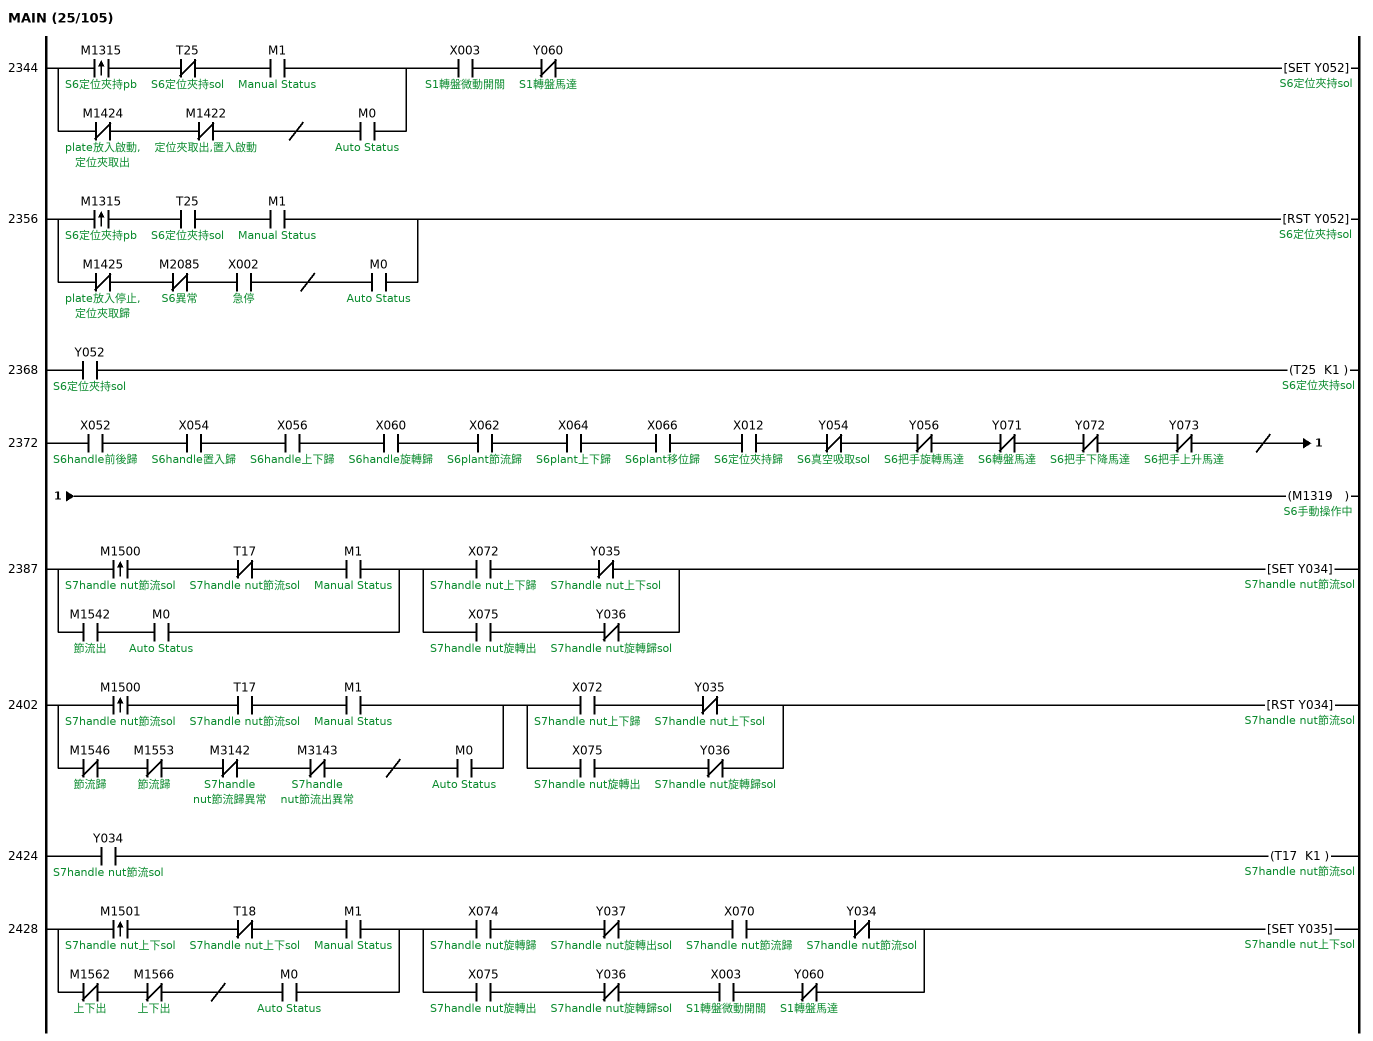
[picture p24: ladder of MAIN, rungs at steps 2344 to 2428]
2344  LDP     M1315  ; S6定位夾持pb
      ANI     T25  ; S6定位夾持sol
      AND     M1  ; Manual Status
      LDI     M1424  ; plate放入啟動,定位夾取出
      ANI     M1422  ; 定位夾取出,置入啟動
      INV
      AND     M0  ; Auto Status
      ORB
      AND     X003  ; S1轉盤微動開關
      ANI     Y060  ; S1轉盤馬達
      SET     Y052  ; S6定位夾持sol
2356  LDP     M1315  ; S6定位夾持pb
      AND     T25  ; S6定位夾持sol
      AND     M1  ; Manual Status
      LDI     M1425  ; plate放入停止,定位夾取歸
      ANI     M2085  ; S6異常
      AND     X002  ; 急停
      INV
      AND     M0  ; Auto Status
      ORB
      RST     Y052  ; S6定位夾持sol
2368  LD      Y052  ; S6定位夾持sol
      OUT     T25 K1  ; S6定位夾持sol
2372  LD      X052  ; S6handle前後歸
      AND     X054  ; S6handle置入歸
      AND     X056  ; S6handle上下歸
      AND     X060  ; S6handle旋轉歸
      AND     X062  ; S6plant節流歸
      AND     X064  ; S6plant上下歸
      AND     X066  ; S6plant移位歸
      AND     X012  ; S6定位夾持歸
      ANI     Y054  ; S6真空吸取sol
      ANI     Y056  ; S6把手旋轉馬達
      ANI     Y071  ; S6轉盤馬達
      ANI     Y072  ; S6把手下降馬達
      ANI     Y073  ; S6把手上升馬達
      INV
      OUT     M1319  ; S6手動操作中
2387  LDP     M1500  ; S7handle nut節流sol
      ANI     T17  ; S7handle nut節流sol
      AND     M1  ; Manual Status
      LD      M1542  ; 節流出
      AND     M0  ; Auto Status
      ORB
      LD      X072  ; S7handle nut上下歸
      ANI     Y035  ; S7handle nut上下sol
      LD      X075  ; S7handle nut旋轉出
      ANI     Y036  ; S7handle nut旋轉歸sol
      ORB
      ANB
      SET     Y034  ; S7handle nut節流sol
2402  LDP     M1500  ; S7handle nut節流sol
      AND     T17  ; S7handle nut節流sol
      AND     M1  ; Manual Status
      LDI     M1546  ; 節流歸
      ANI     M1553  ; 節流歸
      ANI     M3142  ; S7handle nut節流歸異常
      ANI     M3143  ; S7handle nut節流出異常
      INV
      AND     M0  ; Auto Status
      ORB
      LD      X072  ; S7handle nut上下歸
      ANI     Y035  ; S7handle nut上下sol
      LD      X075  ; S7handle nut旋轉出
      ANI     Y036  ; S7handle nut旋轉歸sol
      ORB
      ANB
      RST     Y034  ; S7handle nut節流sol
2424  LD      Y034  ; S7handle nut節流sol
      OUT     T17 K1  ; S7handle nut節流sol
2428  LDP     M1501  ; S7handle nut上下sol
      ANI     T18  ; S7handle nut上下sol
      AND     M1  ; Manual Status
      LDI     M1562  ; 上下出
      ANI     M1566  ; 上下出
      INV
      AND     M0  ; Auto Status
      ORB
      LD      X074  ; S7handle nut旋轉歸
      ANI     Y037  ; S7handle nut旋轉出sol
      AND     X070  ; S7handle nut節流歸
      ANI     Y034  ; S7handle nut節流sol
      LD      X075  ; S7handle nut旋轉出
      ANI     Y036  ; S7handle nut旋轉歸sol
      AND     X003  ; S1轉盤微動開關
      ANI     Y060  ; S1轉盤馬達
      ORB
      ANB
      SET     Y035  ; S7handle nut上下sol
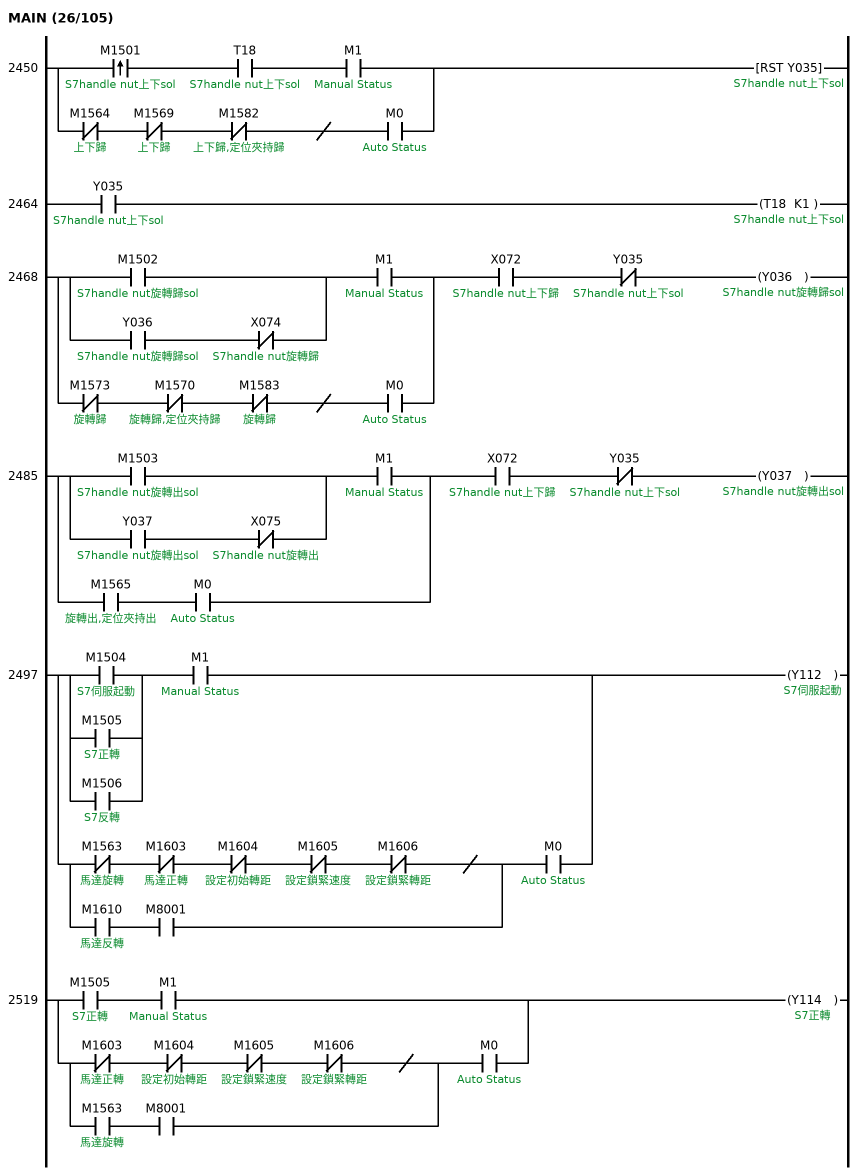
2450  LDP     M1501  ; S7handle nut上下sol
      AND     T18  ; S7handle nut上下sol
      AND     M1  ; Manual Status
      LDI     M1564  ; 上下歸
      ANI     M1569  ; 上下歸
      ANI     M1582  ; 上下歸,定位夾持歸
      INV
      AND     M0  ; Auto Status
      ORB
      RST     Y035  ; S7handle nut上下sol
2464  LD      Y035  ; S7handle nut上下sol
      OUT     T18 K1  ; S7handle nut上下sol
2468  LD      M1502  ; S7handle nut旋轉歸sol
      LD      Y036  ; S7handle nut旋轉歸sol
      ANI     X074  ; S7handle nut旋轉歸
      ORB
      AND     M1  ; Manual Status
      LDI     M1573  ; 旋轉歸
      ANI     M1570  ; 旋轉歸,定位夾持歸
      ANI     M1583  ; 旋轉歸
      INV
      AND     M0  ; Auto Status
      ORB
      AND     X072  ; S7handle nut上下歸
      ANI     Y035  ; S7handle nut上下sol
      OUT     Y036  ; S7handle nut旋轉歸sol
2485  LD      M1503  ; S7handle nut旋轉出sol
      LD      Y037  ; S7handle nut旋轉出sol
      ANI     X075  ; S7handle nut旋轉出
      ORB
      AND     M1  ; Manual Status
      LD      M1565  ; 旋轉出,定位夾持出
      AND     M0  ; Auto Status
      ORB
      AND     X072  ; S7handle nut上下歸
      ANI     Y035  ; S7handle nut上下sol
      OUT     Y037  ; S7handle nut旋轉出sol
2497  LD      M1504  ; S7伺服起動
      OR      M1505  ; S7正轉
      OR      M1506  ; S7反轉
      AND     M1  ; Manual Status
      LDI     M1563  ; 馬達旋轉
      ANI     M1603  ; 馬達正轉
      ANI     M1604  ; 設定初始轉距
      ANI     M1605  ; 設定鎖緊速度
      ANI     M1606  ; 設定鎖緊轉距
      INV
      LD      M1610  ; 馬達反轉
      AND     M8001
      ORB
      AND     M0  ; Auto Status
      ORB
      OUT     Y112  ; S7伺服起動
2519  LD      M1505  ; S7正轉
      AND     M1  ; Manual Status
      LDI     M1603  ; 馬達正轉
      ANI     M1604  ; 設定初始轉距
      ANI     M1605  ; 設定鎖緊速度
      ANI     M1606  ; 設定鎖緊轉距
      INV
      LD      M1563  ; 馬達旋轉
      AND     M8001
      ORB
      AND     M0  ; Auto Status
      ORB
      OUT     Y114  ; S7正轉
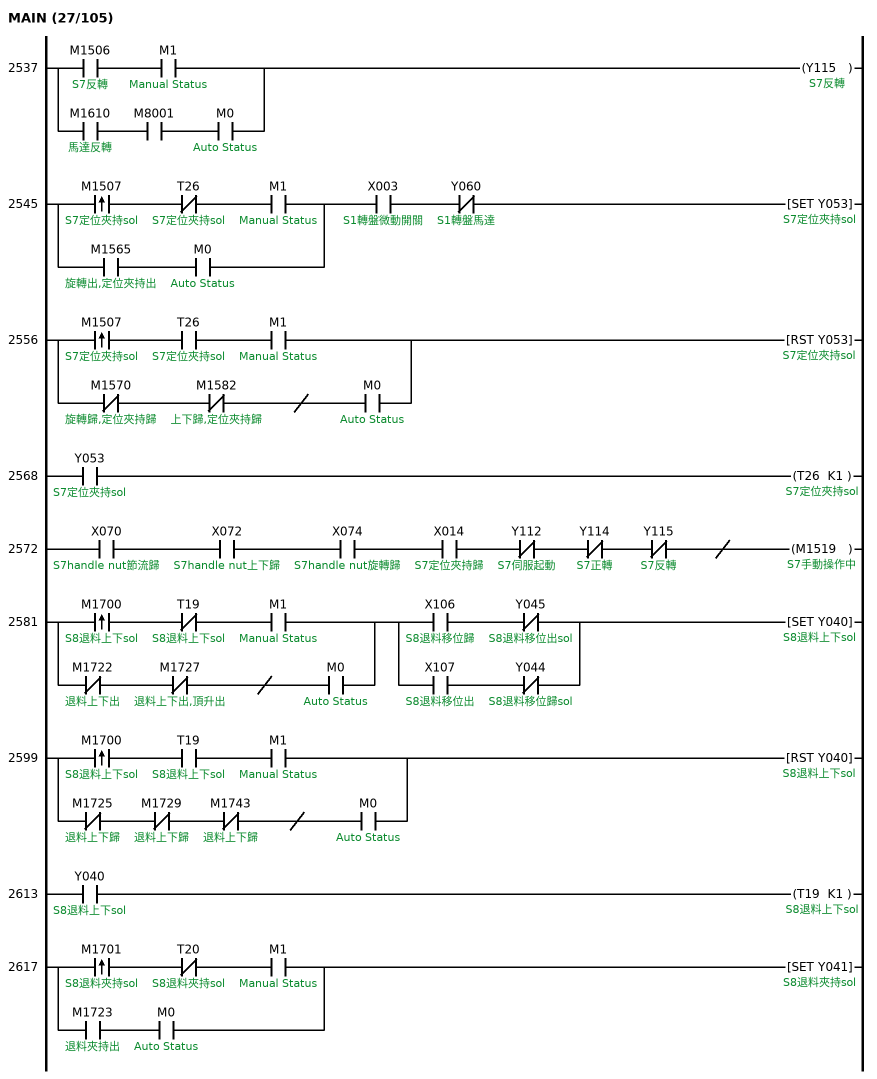
2537  LD      M1506  ; S7反轉
      AND     M1  ; Manual Status
      LD      M1610  ; 馬達反轉
      AND     M8001
      AND     M0  ; Auto Status
      ORB
      OUT     Y115  ; S7反轉
2545  LDP     M1507  ; S7定位夾持sol
      ANI     T26  ; S7定位夾持sol
      AND     M1  ; Manual Status
      LD      M1565  ; 旋轉出,定位夾持出
      AND     M0  ; Auto Status
      ORB
      AND     X003  ; S1轉盤微動開關
      ANI     Y060  ; S1轉盤馬達
      SET     Y053  ; S7定位夾持sol
2556  LDP     M1507  ; S7定位夾持sol
      AND     T26  ; S7定位夾持sol
      AND     M1  ; Manual Status
      LDI     M1570  ; 旋轉歸,定位夾持歸
      ANI     M1582  ; 上下歸,定位夾持歸
      INV
      AND     M0  ; Auto Status
      ORB
      RST     Y053  ; S7定位夾持sol
2568  LD      Y053  ; S7定位夾持sol
      OUT     T26 K1  ; S7定位夾持sol
2572  LD      X070  ; S7handle nut節流歸
      AND     X072  ; S7handle nut上下歸
      AND     X074  ; S7handle nut旋轉歸
      AND     X014  ; S7定位夾持歸
      ANI     Y112  ; S7伺服起動
      ANI     Y114  ; S7正轉
      ANI     Y115  ; S7反轉
      INV
      OUT     M1519  ; S7手動操作中
2581  LDP     M1700  ; S8退料上下sol
      ANI     T19  ; S8退料上下sol
      AND     M1  ; Manual Status
      LDI     M1722  ; 退料上下出
      ANI     M1727  ; 退料上下出,頂升出
      INV
      AND     M0  ; Auto Status
      ORB
      LD      X106  ; S8退料移位歸
      ANI     Y045  ; S8退料移位出sol
      LD      X107  ; S8退料移位出
      ANI     Y044  ; S8退料移位歸sol
      ORB
      ANB
      SET     Y040  ; S8退料上下sol
2599  LDP     M1700  ; S8退料上下sol
      AND     T19  ; S8退料上下sol
      AND     M1  ; Manual Status
      LDI     M1725  ; 退料上下歸
      ANI     M1729  ; 退料上下歸
      ANI     M1743  ; 退料上下歸
      INV
      AND     M0  ; Auto Status
      ORB
      RST     Y040  ; S8退料上下sol
2613  LD      Y040  ; S8退料上下sol
      OUT     T19 K1  ; S8退料上下sol
2617  LDP     M1701  ; S8退料夾持sol
      ANI     T20  ; S8退料夾持sol
      AND     M1  ; Manual Status
      LD      M1723  ; 退料夾持出
      AND     M0  ; Auto Status
      ORB
      SET     Y041  ; S8退料夾持sol
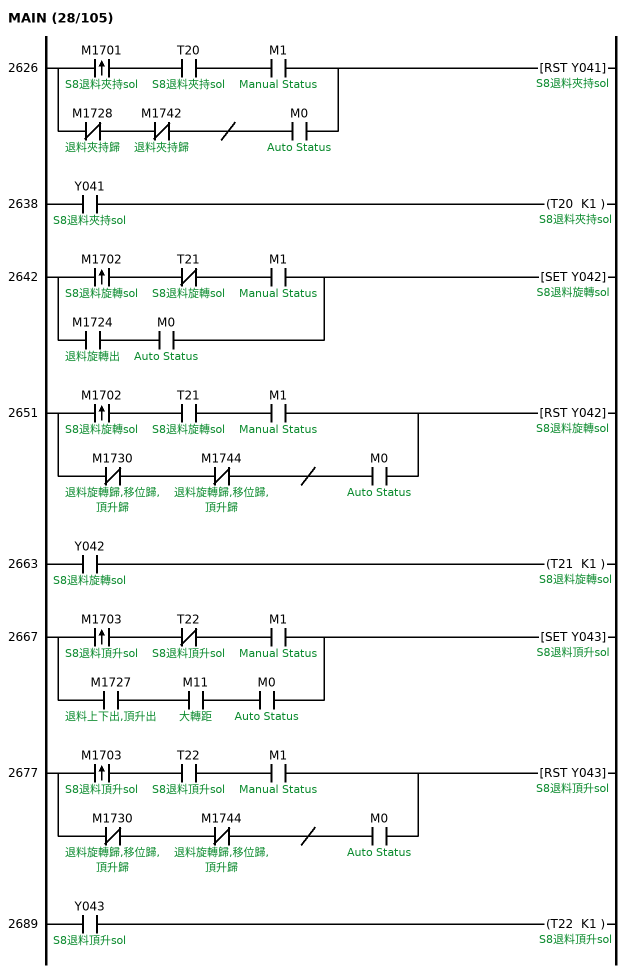
2626  LDP     M1701  ; S8退料夾持sol
      AND     T20  ; S8退料夾持sol
      AND     M1  ; Manual Status
      LDI     M1728  ; 退料夾持歸
      ANI     M1742  ; 退料夾持歸
      INV
      AND     M0  ; Auto Status
      ORB
      RST     Y041  ; S8退料夾持sol
2638  LD      Y041  ; S8退料夾持sol
      OUT     T20 K1  ; S8退料夾持sol
2642  LDP     M1702  ; S8退料旋轉sol
      ANI     T21  ; S8退料旋轉sol
      AND     M1  ; Manual Status
      LD      M1724  ; 退料旋轉出
      AND     M0  ; Auto Status
      ORB
      SET     Y042  ; S8退料旋轉sol
2651  LDP     M1702  ; S8退料旋轉sol
      AND     T21  ; S8退料旋轉sol
      AND     M1  ; Manual Status
      LDI     M1730  ; 退料旋轉歸,移位歸,頂升歸
      ANI     M1744  ; 退料旋轉歸,移位歸,頂升歸
      INV
      AND     M0  ; Auto Status
      ORB
      RST     Y042  ; S8退料旋轉sol
2663  LD      Y042  ; S8退料旋轉sol
      OUT     T21 K1  ; S8退料旋轉sol
2667  LDP     M1703  ; S8退料頂升sol
      ANI     T22  ; S8退料頂升sol
      AND     M1  ; Manual Status
      LD      M1727  ; 退料上下出,頂升出
      AND     M11  ; 大轉距
      AND     M0  ; Auto Status
      ORB
      SET     Y043  ; S8退料頂升sol
2677  LDP     M1703  ; S8退料頂升sol
      AND     T22  ; S8退料頂升sol
      AND     M1  ; Manual Status
      LDI     M1730  ; 退料旋轉歸,移位歸,頂升歸
      ANI     M1744  ; 退料旋轉歸,移位歸,頂升歸
      INV
      AND     M0  ; Auto Status
      ORB
      RST     Y043  ; S8退料頂升sol
2689  LD      Y043  ; S8退料頂升sol
      OUT     T22 K1  ; S8退料頂升sol
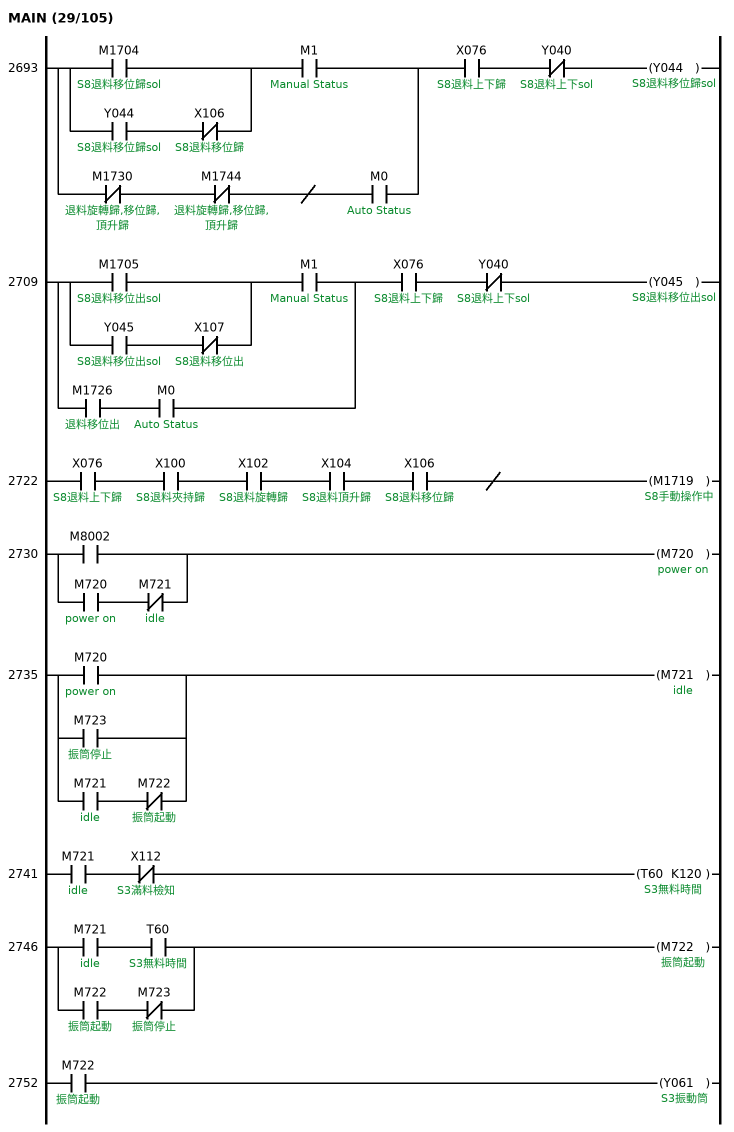
2693  LD      M1704  ; S8退料移位歸sol
      LD      Y044  ; S8退料移位歸sol
      ANI     X106  ; S8退料移位歸
      ORB
      AND     M1  ; Manual Status
      LDI     M1730  ; 退料旋轉歸,移位歸,頂升歸
      ANI     M1744  ; 退料旋轉歸,移位歸,頂升歸
      INV
      AND     M0  ; Auto Status
      ORB
      AND     X076  ; S8退料上下歸
      ANI     Y040  ; S8退料上下sol
      OUT     Y044  ; S8退料移位歸sol
2709  LD      M1705  ; S8退料移位出sol
      LD      Y045  ; S8退料移位出sol
      ANI     X107  ; S8退料移位出
      ORB
      AND     M1  ; Manual Status
      LD      M1726  ; 退料移位出
      AND     M0  ; Auto Status
      ORB
      AND     X076  ; S8退料上下歸
      ANI     Y040  ; S8退料上下sol
      OUT     Y045  ; S8退料移位出sol
2722  LD      X076  ; S8退料上下歸
      AND     X100  ; S8退料夾持歸
      AND     X102  ; S8退料旋轉歸
      AND     X104  ; S8退料頂升歸
      AND     X106  ; S8退料移位歸
      INV
      OUT     M1719  ; S8手動操作中
2730  LD      M8002
      LD      M720  ; power on
      ANI     M721  ; idle
      ORB
      OUT     M720  ; power on
2735  LD      M720  ; power on
      OR      M723  ; 振筒停止
      LD      M721  ; idle
      ANI     M722  ; 振筒起動
      ORB
      OUT     M721  ; idle
2741  LD      M721  ; idle
      ANI     X112  ; S3滿料檢知
      OUT     T60 K120  ; S3無料時間
2746  LD      M721  ; idle
      AND     T60  ; S3無料時間
      LD      M722  ; 振筒起動
      ANI     M723  ; 振筒停止
      ORB
      OUT     M722  ; 振筒起動
2752  LD      M722  ; 振筒起動
      OUT     Y061  ; S3振動筒
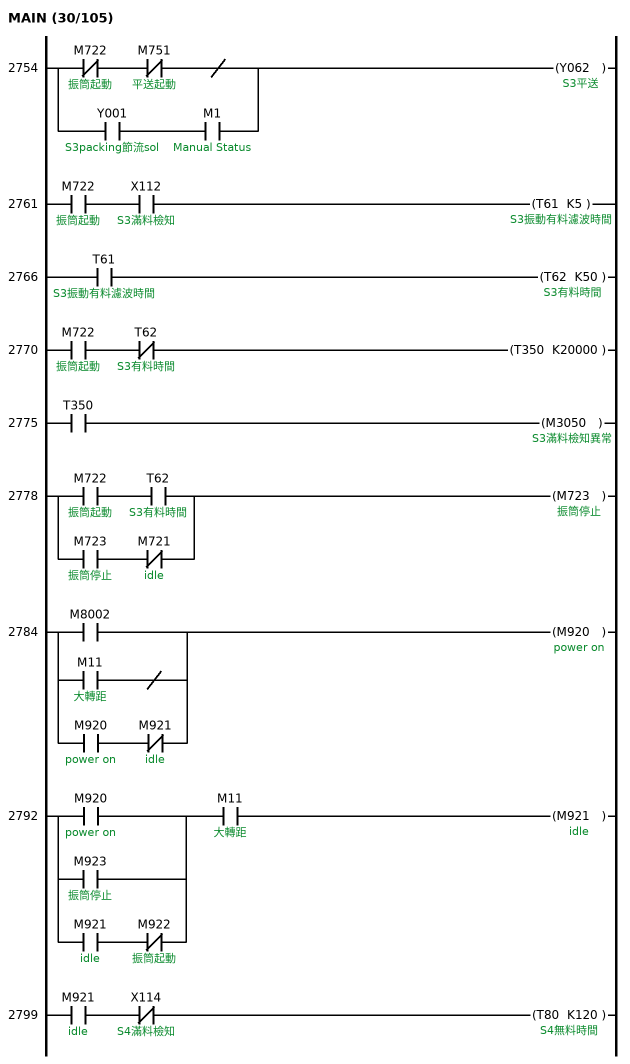
2754  LDI     M722  ; 振筒起動
      ANI     M751  ; 平送起動
      INV
      LD      Y001  ; S3packing節流sol
      AND     M1  ; Manual Status
      ORB
      OUT     Y062  ; S3平送
2761  LD      M722  ; 振筒起動
      AND     X112  ; S3滿料檢知
      OUT     T61 K5  ; S3振動有料濾波時間
2766  LD      T61  ; S3振動有料濾波時間
      OUT     T62 K50  ; S3有料時間
2770  LD      M722  ; 振筒起動
      ANI     T62  ; S3有料時間
      OUT     T350 K20000
2775  LD      T350
      OUT     M3050  ; S3滿料檢知異常
2778  LD      M722  ; 振筒起動
      AND     T62  ; S3有料時間
      LD      M723  ; 振筒停止
      ANI     M721  ; idle
      ORB
      OUT     M723  ; 振筒停止
2784  LD      M8002
      LD      M11  ; 大轉距
      INV
      ORB
      LD      M920  ; power on
      ANI     M921  ; idle
      ORB
      OUT     M920  ; power on
2792  LD      M920  ; power on
      OR      M923  ; 振筒停止
      LD      M921  ; idle
      ANI     M922  ; 振筒起動
      ORB
      AND     M11  ; 大轉距
      OUT     M921  ; idle
2799  LD      M921  ; idle
      ANI     X114  ; S4滿料檢知
      OUT     T80 K120  ; S4無料時間
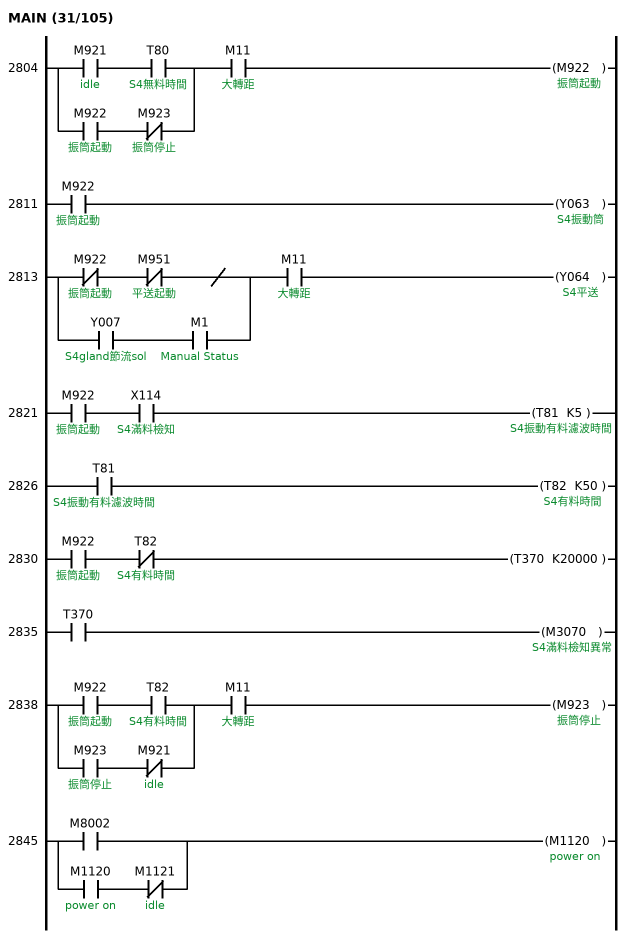
2804  LD      M921  ; idle
      AND     T80  ; S4無料時間
      LD      M922  ; 振筒起動
      ANI     M923  ; 振筒停止
      ORB
      AND     M11  ; 大轉距
      OUT     M922  ; 振筒起動
2811  LD      M922  ; 振筒起動
      OUT     Y063  ; S4振動筒
2813  LDI     M922  ; 振筒起動
      ANI     M951  ; 平送起動
      INV
      LD      Y007  ; S4gland節流sol
      AND     M1  ; Manual Status
      ORB
      AND     M11  ; 大轉距
      OUT     Y064  ; S4平送
2821  LD      M922  ; 振筒起動
      AND     X114  ; S4滿料檢知
      OUT     T81 K5  ; S4振動有料濾波時間
2826  LD      T81  ; S4振動有料濾波時間
      OUT     T82 K50  ; S4有料時間
2830  LD      M922  ; 振筒起動
      ANI     T82  ; S4有料時間
      OUT     T370 K20000
2835  LD      T370
      OUT     M3070  ; S4滿料檢知異常
2838  LD      M922  ; 振筒起動
      AND     T82  ; S4有料時間
      LD      M923  ; 振筒停止
      ANI     M921  ; idle
      ORB
      AND     M11  ; 大轉距
      OUT     M923  ; 振筒停止
2845  LD      M8002
      LD      M1120  ; power on
      ANI     M1121  ; idle
      ORB
      OUT     M1120  ; power on
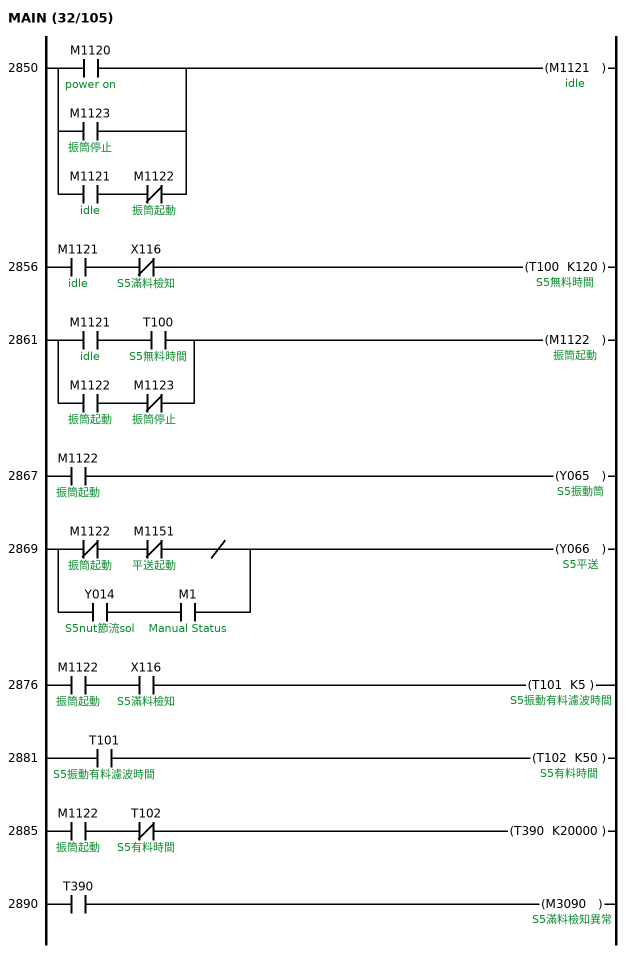
2850  LD      M1120  ; power on
      OR      M1123  ; 振筒停止
      LD      M1121  ; idle
      ANI     M1122  ; 振筒起動
      ORB
      OUT     M1121  ; idle
2856  LD      M1121  ; idle
      ANI     X116  ; S5滿料檢知
      OUT     T100 K120  ; S5無料時間
2861  LD      M1121  ; idle
      AND     T100  ; S5無料時間
      LD      M1122  ; 振筒起動
      ANI     M1123  ; 振筒停止
      ORB
      OUT     M1122  ; 振筒起動
2867  LD      M1122  ; 振筒起動
      OUT     Y065  ; S5振動筒
2869  LDI     M1122  ; 振筒起動
      ANI     M1151  ; 平送起動
      INV
      LD      Y014  ; S5nut節流sol
      AND     M1  ; Manual Status
      ORB
      OUT     Y066  ; S5平送
2876  LD      M1122  ; 振筒起動
      AND     X116  ; S5滿料檢知
      OUT     T101 K5  ; S5振動有料濾波時間
2881  LD      T101  ; S5振動有料濾波時間
      OUT     T102 K50  ; S5有料時間
2885  LD      M1122  ; 振筒起動
      ANI     T102  ; S5有料時間
      OUT     T390 K20000
2890  LD      T390
      OUT     M3090  ; S5滿料檢知異常
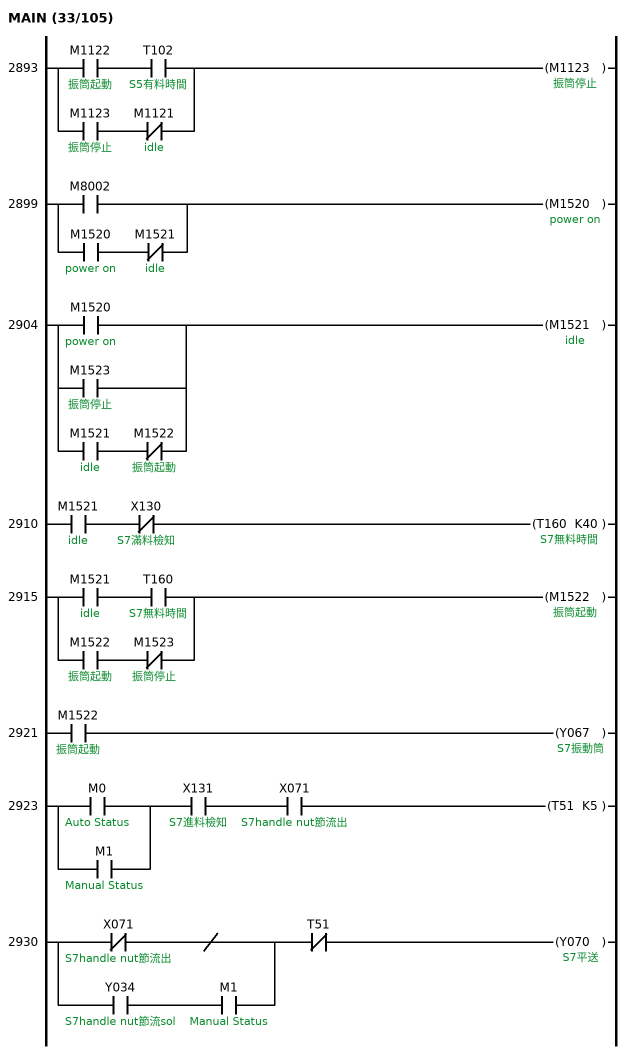
2893  LD      M1122  ; 振筒起動
      AND     T102  ; S5有料時間
      LD      M1123  ; 振筒停止
      ANI     M1121  ; idle
      ORB
      OUT     M1123  ; 振筒停止
2899  LD      M8002
      LD      M1520  ; power on
      ANI     M1521  ; idle
      ORB
      OUT     M1520  ; power on
2904  LD      M1520  ; power on
      OR      M1523  ; 振筒停止
      LD      M1521  ; idle
      ANI     M1522  ; 振筒起動
      ORB
      OUT     M1521  ; idle
2910  LD      M1521  ; idle
      ANI     X130  ; S7滿料檢知
      OUT     T160 K40  ; S7無料時間
2915  LD      M1521  ; idle
      AND     T160  ; S7無料時間
      LD      M1522  ; 振筒起動
      ANI     M1523  ; 振筒停止
      ORB
      OUT     M1522  ; 振筒起動
2921  LD      M1522  ; 振筒起動
      OUT     Y067  ; S7振動筒
2923  LD      M0  ; Auto Status
      OR      M1  ; Manual Status
      AND     X131  ; S7進料檢知
      AND     X071  ; S7handle nut節流出
      OUT     T51 K5
2930  LDI     X071  ; S7handle nut節流出
      INV
      LD      Y034  ; S7handle nut節流sol
      AND     M1  ; Manual Status
      ORB
      ANI     T51
      OUT     Y070  ; S7平送
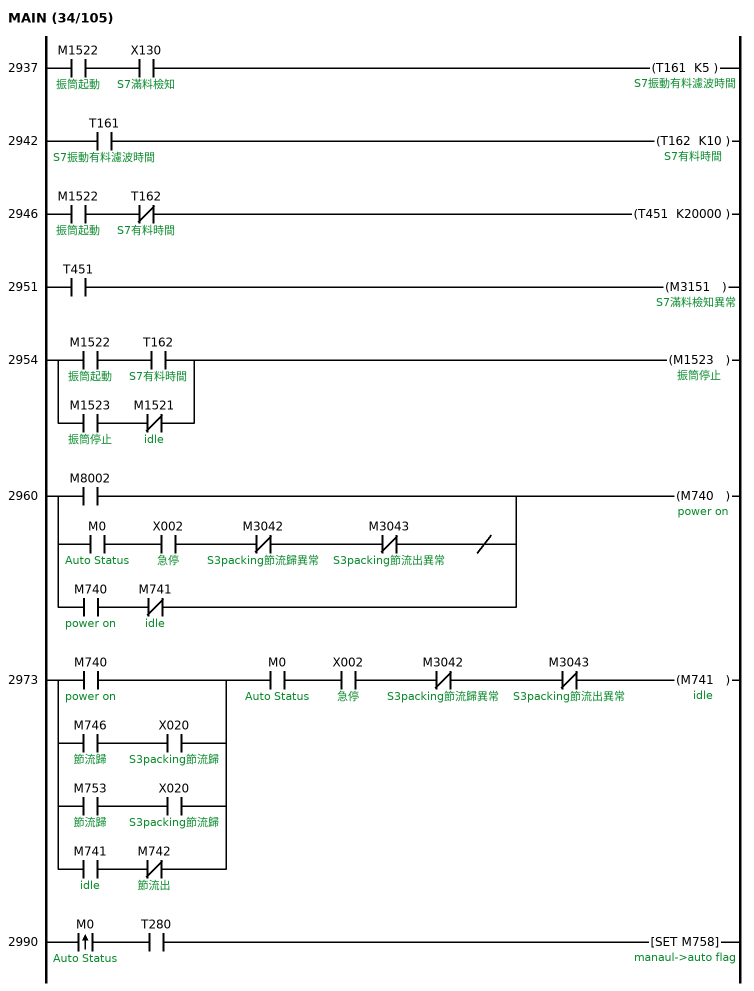
2937  LD      M1522  ; 振筒起動
      AND     X130  ; S7滿料檢知
      OUT     T161 K5  ; S7振動有料濾波時間
2942  LD      T161  ; S7振動有料濾波時間
      OUT     T162 K10  ; S7有料時間
2946  LD      M1522  ; 振筒起動
      ANI     T162  ; S7有料時間
      OUT     T451 K20000
2951  LD      T451
      OUT     M3151  ; S7滿料檢知異常
2954  LD      M1522  ; 振筒起動
      AND     T162  ; S7有料時間
      LD      M1523  ; 振筒停止
      ANI     M1521  ; idle
      ORB
      OUT     M1523  ; 振筒停止
2960  LD      M8002
      LD      M0  ; Auto Status
      AND     X002  ; 急停
      ANI     M3042  ; S3packing節流歸異常
      ANI     M3043  ; S3packing節流出異常
      INV
      ORB
      LD      M740  ; power on
      ANI     M741  ; idle
      ORB
      OUT     M740  ; power on
2973  LD      M740  ; power on
      LD      M746  ; 節流歸
      AND     X020  ; S3packing節流歸
      ORB
      LD      M753  ; 節流歸
      AND     X020  ; S3packing節流歸
      ORB
      LD      M741  ; idle
      ANI     M742  ; 節流出
      ORB
      AND     M0  ; Auto Status
      AND     X002  ; 急停
      ANI     M3042  ; S3packing節流歸異常
      ANI     M3043  ; S3packing節流出異常
      OUT     M741  ; idle
2990  LDP     M0  ; Auto Status
      AND     T280
      SET     M758  ; manaul->auto flag
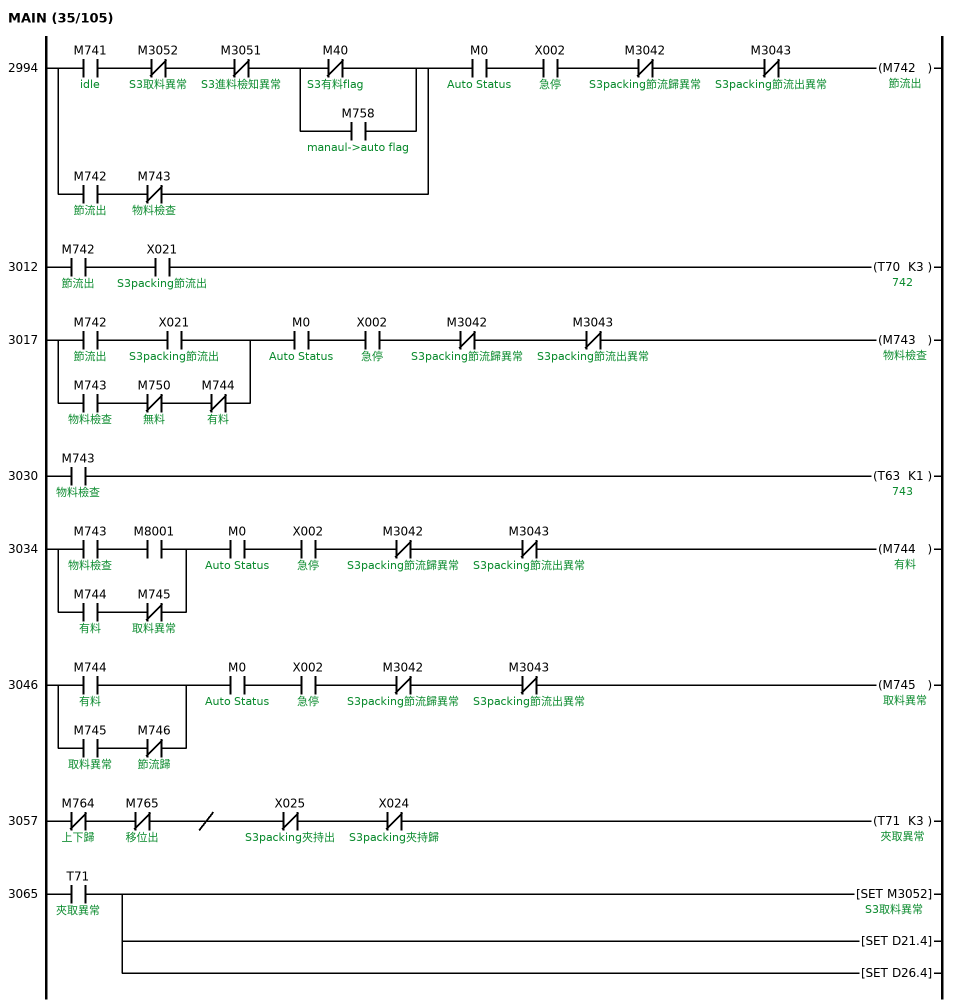
2994  LD      M741  ; idle
      ANI     M3052  ; S3取料異常
      ANI     M3051  ; S3進料檢知異常
      LDI     M40  ; S3有料flag
      OR      M758  ; manaul->auto flag
      ANB
      LD      M742  ; 節流出
      ANI     M743  ; 物料檢查
      ORB
      AND     M0  ; Auto Status
      AND     X002  ; 急停
      ANI     M3042  ; S3packing節流歸異常
      ANI     M3043  ; S3packing節流出異常
      OUT     M742  ; 節流出
3012  LD      M742  ; 節流出
      AND     X021  ; S3packing節流出
      OUT     T70 K3  ; 742
3017  LD      M742  ; 節流出
      AND     X021  ; S3packing節流出
      LD      M743  ; 物料檢查
      ANI     M750  ; 無料
      ANI     M744  ; 有料
      ORB
      AND     M0  ; Auto Status
      AND     X002  ; 急停
      ANI     M3042  ; S3packing節流歸異常
      ANI     M3043  ; S3packing節流出異常
      OUT     M743  ; 物料檢查
3030  LD      M743  ; 物料檢查
      OUT     T63 K1  ; 743
3034  LD      M743  ; 物料檢查
      AND     M8001
      LD      M744  ; 有料
      ANI     M745  ; 取料異常
      ORB
      AND     M0  ; Auto Status
      AND     X002  ; 急停
      ANI     M3042  ; S3packing節流歸異常
      ANI     M3043  ; S3packing節流出異常
      OUT     M744  ; 有料
3046  LD      M744  ; 有料
      LD      M745  ; 取料異常
      ANI     M746  ; 節流歸
      ORB
      AND     M0  ; Auto Status
      AND     X002  ; 急停
      ANI     M3042  ; S3packing節流歸異常
      ANI     M3043  ; S3packing節流出異常
      OUT     M745  ; 取料異常
3057  LDI     M764  ; 上下歸
      ANI     M765  ; 移位出
      INV
      ANI     X025  ; S3packing夾持出
      ANI     X024  ; S3packing夾持歸
      OUT     T71 K3  ; 夾取異常
3065  LD      T71  ; 夾取異常
      SET     M3052  ; S3取料異常
      SET     D21.4
      SET     D26.4
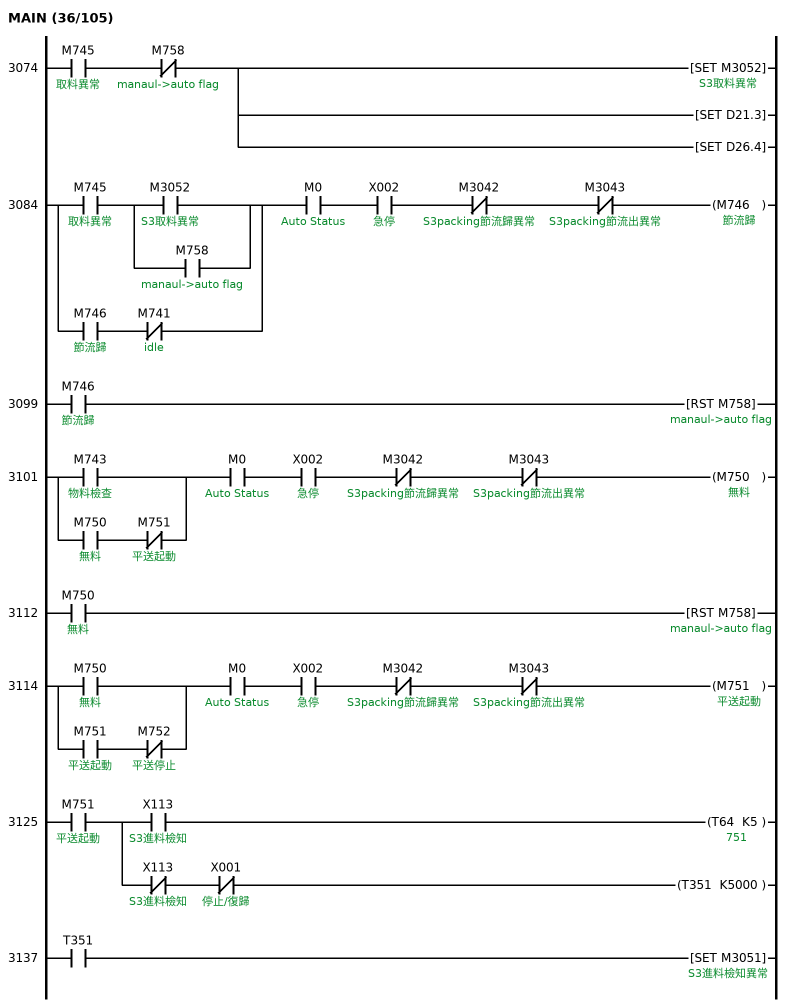
3074  LD      M745  ; 取料異常
      ANI     M758  ; manaul->auto flag
      SET     M3052  ; S3取料異常
      SET     D21.3
      SET     D26.4
3084  LD      M745  ; 取料異常
      LD      M3052  ; S3取料異常
      OR      M758  ; manaul->auto flag
      ANB
      LD      M746  ; 節流歸
      ANI     M741  ; idle
      ORB
      AND     M0  ; Auto Status
      AND     X002  ; 急停
      ANI     M3042  ; S3packing節流歸異常
      ANI     M3043  ; S3packing節流出異常
      OUT     M746  ; 節流歸
3099  LD      M746  ; 節流歸
      RST     M758  ; manaul->auto flag
3101  LD      M743  ; 物料檢查
      LD      M750  ; 無料
      ANI     M751  ; 平送起動
      ORB
      AND     M0  ; Auto Status
      AND     X002  ; 急停
      ANI     M3042  ; S3packing節流歸異常
      ANI     M3043  ; S3packing節流出異常
      OUT     M750  ; 無料
3112  LD      M750  ; 無料
      RST     M758  ; manaul->auto flag
3114  LD      M750  ; 無料
      LD      M751  ; 平送起動
      ANI     M752  ; 平送停止
      ORB
      AND     M0  ; Auto Status
      AND     X002  ; 急停
      ANI     M3042  ; S3packing節流歸異常
      ANI     M3043  ; S3packing節流出異常
      OUT     M751  ; 平送起動
3125  LD      M751  ; 平送起動
      MPS
      AND     X113  ; S3進料檢知
      OUT     T64 K5  ; 751
      MPP
      ANI     X113  ; S3進料檢知
      ANI     X001  ; 停止/復歸
      OUT     T351 K5000
3137  LD      T351
      SET     M3051  ; S3進料檢知異常
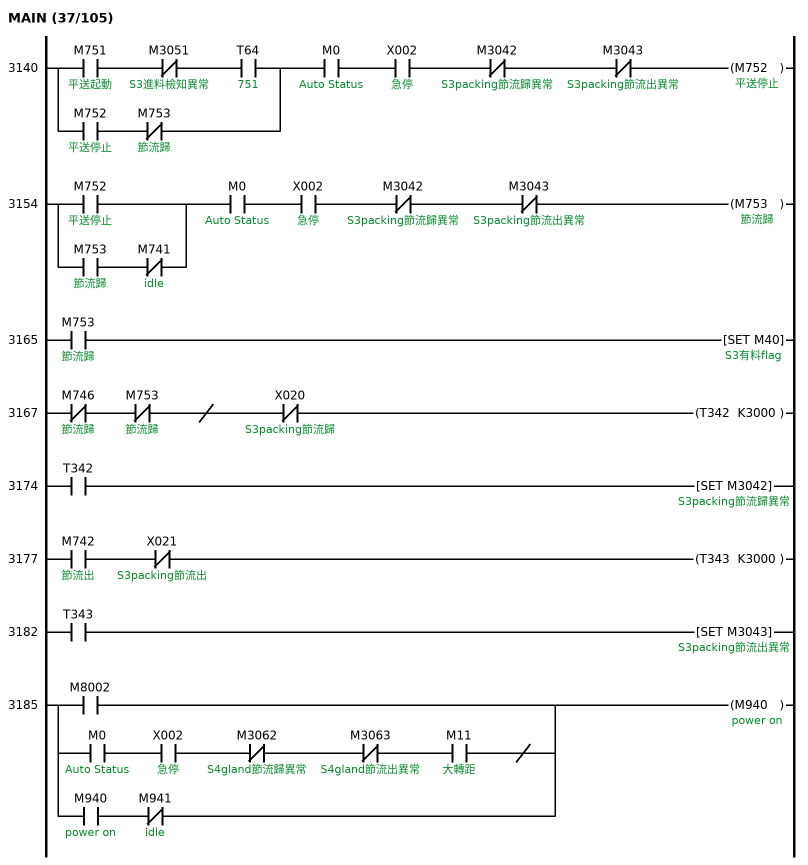
3140  LD      M751  ; 平送起動
      ANI     M3051  ; S3進料檢知異常
      AND     T64  ; 751
      LD      M752  ; 平送停止
      ANI     M753  ; 節流歸
      ORB
      AND     M0  ; Auto Status
      AND     X002  ; 急停
      ANI     M3042  ; S3packing節流歸異常
      ANI     M3043  ; S3packing節流出異常
      OUT     M752  ; 平送停止
3154  LD      M752  ; 平送停止
      LD      M753  ; 節流歸
      ANI     M741  ; idle
      ORB
      AND     M0  ; Auto Status
      AND     X002  ; 急停
      ANI     M3042  ; S3packing節流歸異常
      ANI     M3043  ; S3packing節流出異常
      OUT     M753  ; 節流歸
3165  LD      M753  ; 節流歸
      SET     M40  ; S3有料flag
3167  LDI     M746  ; 節流歸
      ANI     M753  ; 節流歸
      INV
      ANI     X020  ; S3packing節流歸
      OUT     T342 K3000
3174  LD      T342
      SET     M3042  ; S3packing節流歸異常
3177  LD      M742  ; 節流出
      ANI     X021  ; S3packing節流出
      OUT     T343 K3000
3182  LD      T343
      SET     M3043  ; S3packing節流出異常
3185  LD      M8002
      LD      M0  ; Auto Status
      AND     X002  ; 急停
      ANI     M3062  ; S4gland節流歸異常
      ANI     M3063  ; S4gland節流出異常
      AND     M11  ; 大轉距
      INV
      ORB
      LD      M940  ; power on
      ANI     M941  ; idle
      ORB
      OUT     M940  ; power on
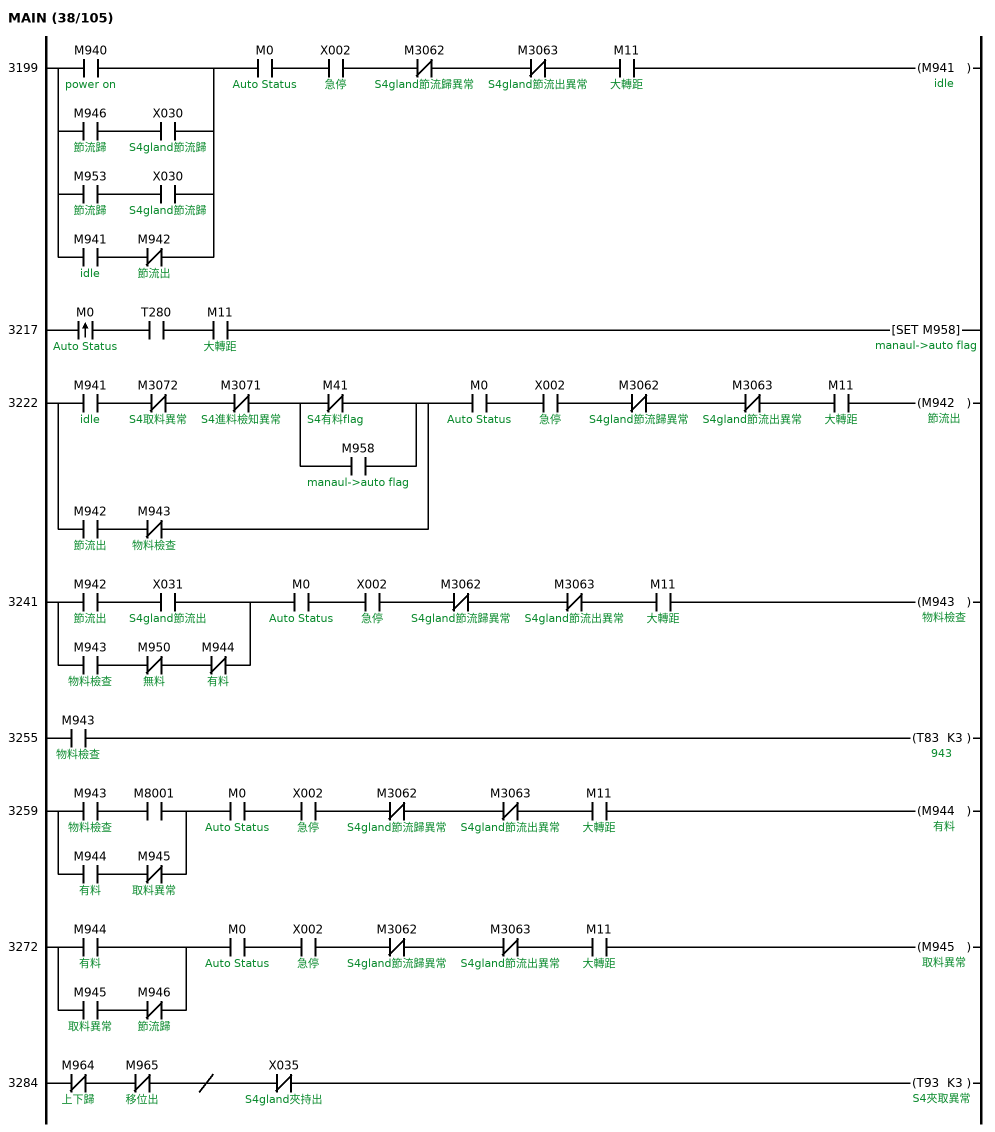
3199  LD      M940  ; power on
      LD      M946  ; 節流歸
      AND     X030  ; S4gland節流歸
      ORB
      LD      M953  ; 節流歸
      AND     X030  ; S4gland節流歸
      ORB
      LD      M941  ; idle
      ANI     M942  ; 節流出
      ORB
      AND     M0  ; Auto Status
      AND     X002  ; 急停
      ANI     M3062  ; S4gland節流歸異常
      ANI     M3063  ; S4gland節流出異常
      AND     M11  ; 大轉距
      OUT     M941  ; idle
3217  LDP     M0  ; Auto Status
      AND     T280
      AND     M11  ; 大轉距
      SET     M958  ; manaul->auto flag
3222  LD      M941  ; idle
      ANI     M3072  ; S4取料異常
      ANI     M3071  ; S4進料檢知異常
      LDI     M41  ; S4有料flag
      OR      M958  ; manaul->auto flag
      ANB
      LD      M942  ; 節流出
      ANI     M943  ; 物料檢查
      ORB
      AND     M0  ; Auto Status
      AND     X002  ; 急停
      ANI     M3062  ; S4gland節流歸異常
      ANI     M3063  ; S4gland節流出異常
      AND     M11  ; 大轉距
      OUT     M942  ; 節流出
3241  LD      M942  ; 節流出
      AND     X031  ; S4gland節流出
      LD      M943  ; 物料檢查
      ANI     M950  ; 無料
      ANI     M944  ; 有料
      ORB
      AND     M0  ; Auto Status
      AND     X002  ; 急停
      ANI     M3062  ; S4gland節流歸異常
      ANI     M3063  ; S4gland節流出異常
      AND     M11  ; 大轉距
      OUT     M943  ; 物料檢查
3255  LD      M943  ; 物料檢查
      OUT     T83 K3  ; 943
3259  LD      M943  ; 物料檢查
      AND     M8001
      LD      M944  ; 有料
      ANI     M945  ; 取料異常
      ORB
      AND     M0  ; Auto Status
      AND     X002  ; 急停
      ANI     M3062  ; S4gland節流歸異常
      ANI     M3063  ; S4gland節流出異常
      AND     M11  ; 大轉距
      OUT     M944  ; 有料
3272  LD      M944  ; 有料
      LD      M945  ; 取料異常
      ANI     M946  ; 節流歸
      ORB
      AND     M0  ; Auto Status
      AND     X002  ; 急停
      ANI     M3062  ; S4gland節流歸異常
      ANI     M3063  ; S4gland節流出異常
      AND     M11  ; 大轉距
      OUT     M945  ; 取料異常
3284  LDI     M964  ; 上下歸
      ANI     M965  ; 移位出
      INV
      ANI     X035  ; S4gland夾持出
      OUT     T93 K3  ; S4夾取異常
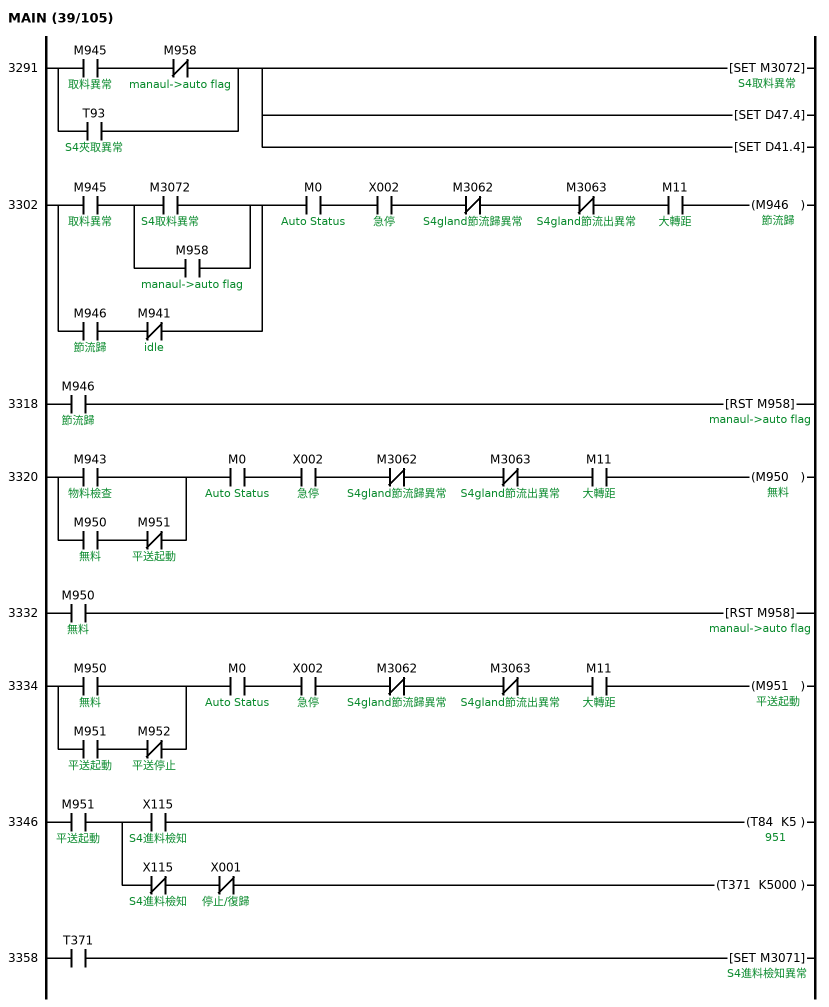
3291  LD      M945  ; 取料異常
      ANI     M958  ; manaul->auto flag
      OR      T93  ; S4夾取異常
      SET     M3072  ; S4取料異常
      SET     D47.4
      SET     D41.4
3302  LD      M945  ; 取料異常
      LD      M3072  ; S4取料異常
      OR      M958  ; manaul->auto flag
      ANB
      LD      M946  ; 節流歸
      ANI     M941  ; idle
      ORB
      AND     M0  ; Auto Status
      AND     X002  ; 急停
      ANI     M3062  ; S4gland節流歸異常
      ANI     M3063  ; S4gland節流出異常
      AND     M11  ; 大轉距
      OUT     M946  ; 節流歸
3318  LD      M946  ; 節流歸
      RST     M958  ; manaul->auto flag
3320  LD      M943  ; 物料檢查
      LD      M950  ; 無料
      ANI     M951  ; 平送起動
      ORB
      AND     M0  ; Auto Status
      AND     X002  ; 急停
      ANI     M3062  ; S4gland節流歸異常
      ANI     M3063  ; S4gland節流出異常
      AND     M11  ; 大轉距
      OUT     M950  ; 無料
3332  LD      M950  ; 無料
      RST     M958  ; manaul->auto flag
3334  LD      M950  ; 無料
      LD      M951  ; 平送起動
      ANI     M952  ; 平送停止
      ORB
      AND     M0  ; Auto Status
      AND     X002  ; 急停
      ANI     M3062  ; S4gland節流歸異常
      ANI     M3063  ; S4gland節流出異常
      AND     M11  ; 大轉距
      OUT     M951  ; 平送起動
3346  LD      M951  ; 平送起動
      MPS
      AND     X115  ; S4進料檢知
      OUT     T84 K5  ; 951
      MPP
      ANI     X115  ; S4進料檢知
      ANI     X001  ; 停止/復歸
      OUT     T371 K5000
3358  LD      T371
      SET     M3071  ; S4進料檢知異常
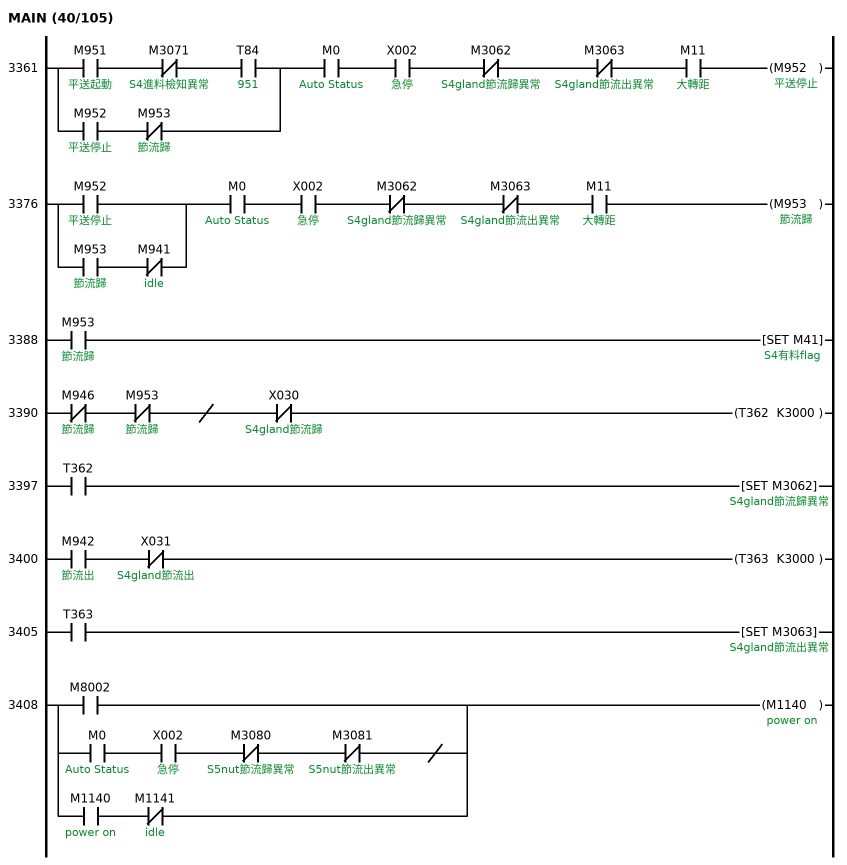
3361  LD      M951  ; 平送起動
      ANI     M3071  ; S4進料檢知異常
      AND     T84  ; 951
      LD      M952  ; 平送停止
      ANI     M953  ; 節流歸
      ORB
      AND     M0  ; Auto Status
      AND     X002  ; 急停
      ANI     M3062  ; S4gland節流歸異常
      ANI     M3063  ; S4gland節流出異常
      AND     M11  ; 大轉距
      OUT     M952  ; 平送停止
3376  LD      M952  ; 平送停止
      LD      M953  ; 節流歸
      ANI     M941  ; idle
      ORB
      AND     M0  ; Auto Status
      AND     X002  ; 急停
      ANI     M3062  ; S4gland節流歸異常
      ANI     M3063  ; S4gland節流出異常
      AND     M11  ; 大轉距
      OUT     M953  ; 節流歸
3388  LD      M953  ; 節流歸
      SET     M41  ; S4有料flag
3390  LDI     M946  ; 節流歸
      ANI     M953  ; 節流歸
      INV
      ANI     X030  ; S4gland節流歸
      OUT     T362 K3000
3397  LD      T362
      SET     M3062  ; S4gland節流歸異常
3400  LD      M942  ; 節流出
      ANI     X031  ; S4gland節流出
      OUT     T363 K3000
3405  LD      T363
      SET     M3063  ; S4gland節流出異常
3408  LD      M8002
      LD      M0  ; Auto Status
      AND     X002  ; 急停
      ANI     M3080  ; S5nut節流歸異常
      ANI     M3081  ; S5nut節流出異常
      INV
      ORB
      LD      M1140  ; power on
      ANI     M1141  ; idle
      ORB
      OUT     M1140  ; power on
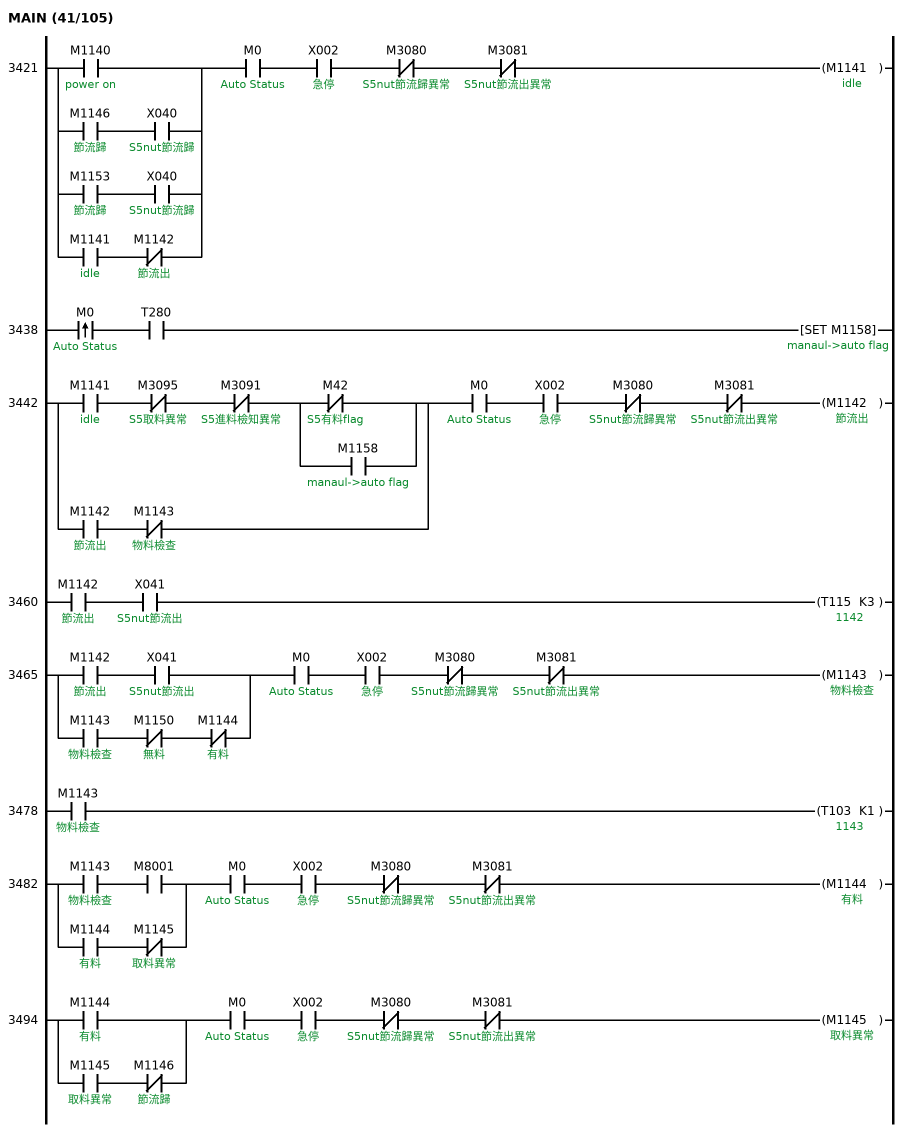
3421  LD      M1140  ; power on
      LD      M1146  ; 節流歸
      AND     X040  ; S5nut節流歸
      ORB
      LD      M1153  ; 節流歸
      AND     X040  ; S5nut節流歸
      ORB
      LD      M1141  ; idle
      ANI     M1142  ; 節流出
      ORB
      AND     M0  ; Auto Status
      AND     X002  ; 急停
      ANI     M3080  ; S5nut節流歸異常
      ANI     M3081  ; S5nut節流出異常
      OUT     M1141  ; idle
3438  LDP     M0  ; Auto Status
      AND     T280
      SET     M1158  ; manaul->auto flag
3442  LD      M1141  ; idle
      ANI     M3095  ; S5取料異常
      ANI     M3091  ; S5進料檢知異常
      LDI     M42  ; S5有料flag
      OR      M1158  ; manaul->auto flag
      ANB
      LD      M1142  ; 節流出
      ANI     M1143  ; 物料檢查
      ORB
      AND     M0  ; Auto Status
      AND     X002  ; 急停
      ANI     M3080  ; S5nut節流歸異常
      ANI     M3081  ; S5nut節流出異常
      OUT     M1142  ; 節流出
3460  LD      M1142  ; 節流出
      AND     X041  ; S5nut節流出
      OUT     T115 K3  ; 1142
3465  LD      M1142  ; 節流出
      AND     X041  ; S5nut節流出
      LD      M1143  ; 物料檢查
      ANI     M1150  ; 無料
      ANI     M1144  ; 有料
      ORB
      AND     M0  ; Auto Status
      AND     X002  ; 急停
      ANI     M3080  ; S5nut節流歸異常
      ANI     M3081  ; S5nut節流出異常
      OUT     M1143  ; 物料檢查
3478  LD      M1143  ; 物料檢查
      OUT     T103 K1  ; 1143
3482  LD      M1143  ; 物料檢查
      AND     M8001
      LD      M1144  ; 有料
      ANI     M1145  ; 取料異常
      ORB
      AND     M0  ; Auto Status
      AND     X002  ; 急停
      ANI     M3080  ; S5nut節流歸異常
      ANI     M3081  ; S5nut節流出異常
      OUT     M1144  ; 有料
3494  LD      M1144  ; 有料
      LD      M1145  ; 取料異常
      ANI     M1146  ; 節流歸
      ORB
      AND     M0  ; Auto Status
      AND     X002  ; 急停
      ANI     M3080  ; S5nut節流歸異常
      ANI     M3081  ; S5nut節流出異常
      OUT     M1145  ; 取料異常
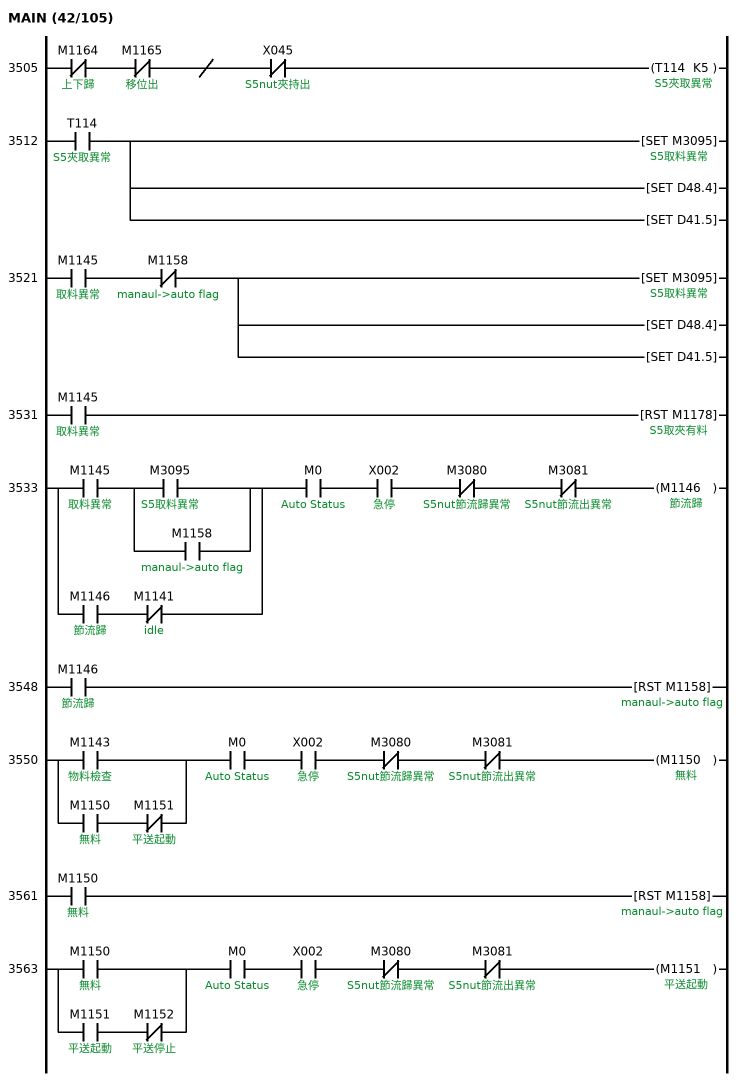
3505  LDI     M1164  ; 上下歸
      ANI     M1165  ; 移位出
      INV
      ANI     X045  ; S5nut夾持出
      OUT     T114 K5  ; S5夾取異常
3512  LD      T114  ; S5夾取異常
      SET     M3095  ; S5取料異常
      SET     D48.4
      SET     D41.5
3521  LD      M1145  ; 取料異常
      ANI     M1158  ; manaul->auto flag
      SET     M3095  ; S5取料異常
      SET     D48.4
      SET     D41.5
3531  LD      M1145  ; 取料異常
      RST     M1178  ; S5取夾有料
3533  LD      M1145  ; 取料異常
      LD      M3095  ; S5取料異常
      OR      M1158  ; manaul->auto flag
      ANB
      LD      M1146  ; 節流歸
      ANI     M1141  ; idle
      ORB
      AND     M0  ; Auto Status
      AND     X002  ; 急停
      ANI     M3080  ; S5nut節流歸異常
      ANI     M3081  ; S5nut節流出異常
      OUT     M1146  ; 節流歸
3548  LD      M1146  ; 節流歸
      RST     M1158  ; manaul->auto flag
3550  LD      M1143  ; 物料檢查
      LD      M1150  ; 無料
      ANI     M1151  ; 平送起動
      ORB
      AND     M0  ; Auto Status
      AND     X002  ; 急停
      ANI     M3080  ; S5nut節流歸異常
      ANI     M3081  ; S5nut節流出異常
      OUT     M1150  ; 無料
3561  LD      M1150  ; 無料
      RST     M1158  ; manaul->auto flag
3563  LD      M1150  ; 無料
      LD      M1151  ; 平送起動
      ANI     M1152  ; 平送停止
      ORB
      AND     M0  ; Auto Status
      AND     X002  ; 急停
      ANI     M3080  ; S5nut節流歸異常
      ANI     M3081  ; S5nut節流出異常
      OUT     M1151  ; 平送起動
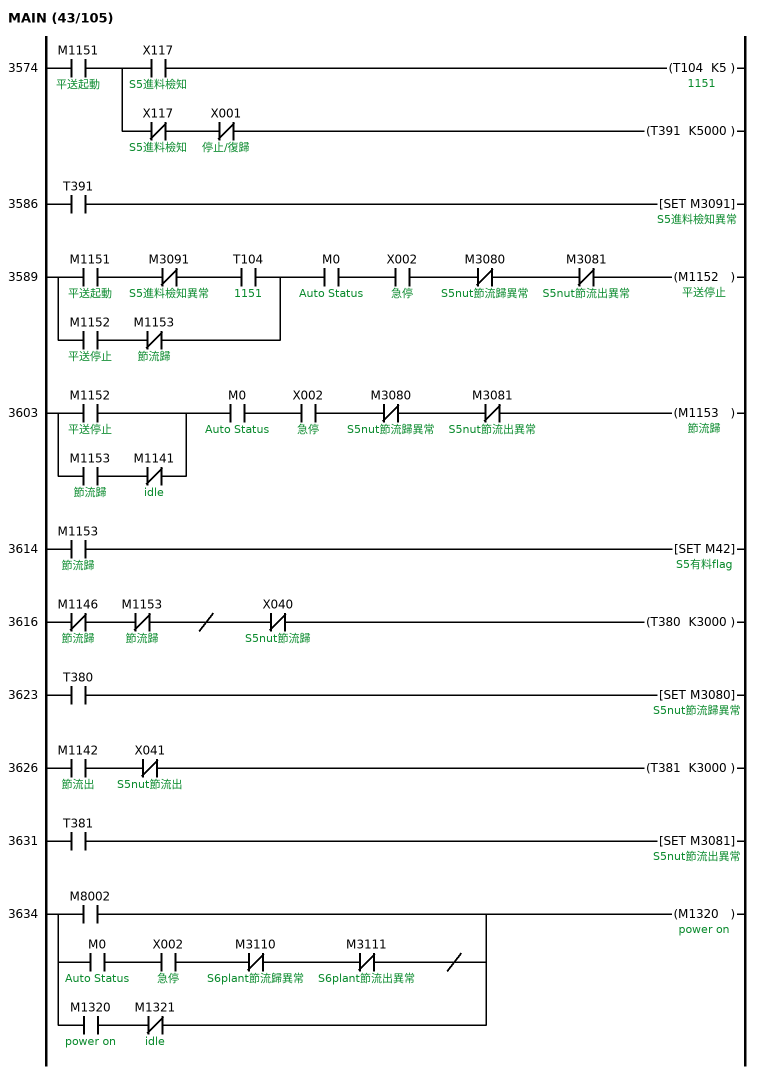
3574  LD      M1151  ; 平送起動
      MPS
      AND     X117  ; S5進料檢知
      OUT     T104 K5  ; 1151
      MPP
      ANI     X117  ; S5進料檢知
      ANI     X001  ; 停止/復歸
      OUT     T391 K5000
3586  LD      T391
      SET     M3091  ; S5進料檢知異常
3589  LD      M1151  ; 平送起動
      ANI     M3091  ; S5進料檢知異常
      AND     T104  ; 1151
      LD      M1152  ; 平送停止
      ANI     M1153  ; 節流歸
      ORB
      AND     M0  ; Auto Status
      AND     X002  ; 急停
      ANI     M3080  ; S5nut節流歸異常
      ANI     M3081  ; S5nut節流出異常
      OUT     M1152  ; 平送停止
3603  LD      M1152  ; 平送停止
      LD      M1153  ; 節流歸
      ANI     M1141  ; idle
      ORB
      AND     M0  ; Auto Status
      AND     X002  ; 急停
      ANI     M3080  ; S5nut節流歸異常
      ANI     M3081  ; S5nut節流出異常
      OUT     M1153  ; 節流歸
3614  LD      M1153  ; 節流歸
      SET     M42  ; S5有料flag
3616  LDI     M1146  ; 節流歸
      ANI     M1153  ; 節流歸
      INV
      ANI     X040  ; S5nut節流歸
      OUT     T380 K3000
3623  LD      T380
      SET     M3080  ; S5nut節流歸異常
3626  LD      M1142  ; 節流出
      ANI     X041  ; S5nut節流出
      OUT     T381 K3000
3631  LD      T381
      SET     M3081  ; S5nut節流出異常
3634  LD      M8002
      LD      M0  ; Auto Status
      AND     X002  ; 急停
      ANI     M3110  ; S6plant節流歸異常
      ANI     M3111  ; S6plant節流出異常
      INV
      ORB
      LD      M1320  ; power on
      ANI     M1321  ; idle
      ORB
      OUT     M1320  ; power on
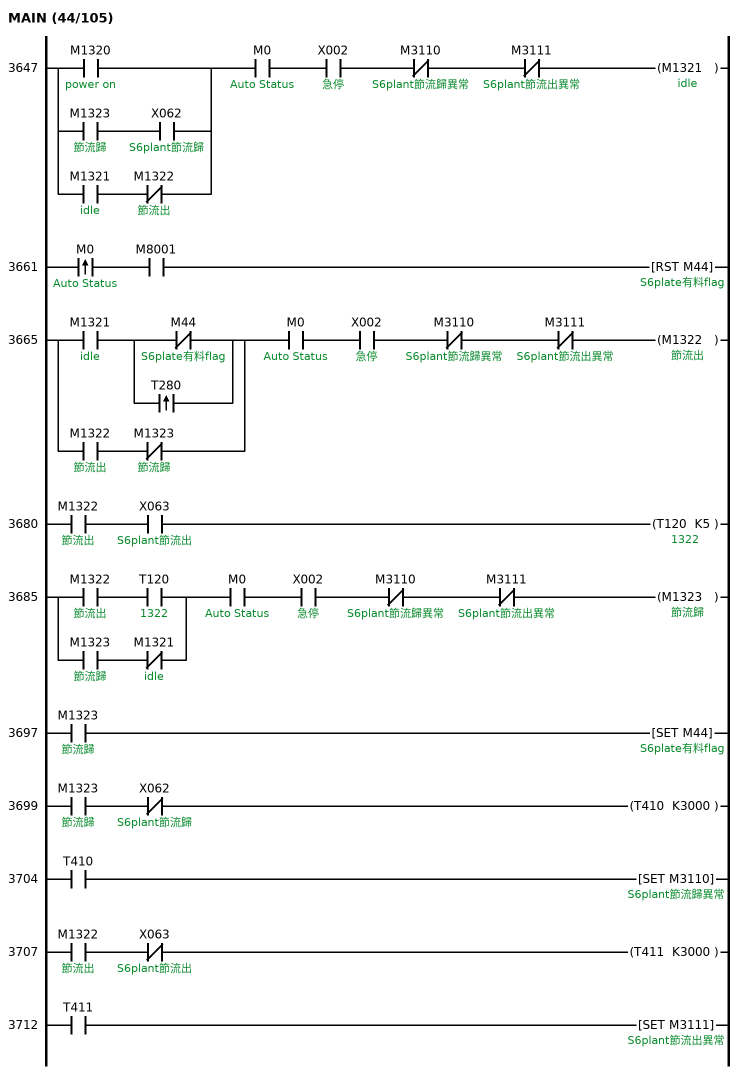
3647  LD      M1320  ; power on
      LD      M1323  ; 節流歸
      AND     X062  ; S6plant節流歸
      ORB
      LD      M1321  ; idle
      ANI     M1322  ; 節流出
      ORB
      AND     M0  ; Auto Status
      AND     X002  ; 急停
      ANI     M3110  ; S6plant節流歸異常
      ANI     M3111  ; S6plant節流出異常
      OUT     M1321  ; idle
3661  LDP     M0  ; Auto Status
      AND     M8001
      RST     M44  ; S6plate有料flag
3665  LD      M1321  ; idle
      LDI     M44  ; S6plate有料flag
      ORP     T280
      ANB
      LD      M1322  ; 節流出
      ANI     M1323  ; 節流歸
      ORB
      AND     M0  ; Auto Status
      AND     X002  ; 急停
      ANI     M3110  ; S6plant節流歸異常
      ANI     M3111  ; S6plant節流出異常
      OUT     M1322  ; 節流出
3680  LD      M1322  ; 節流出
      AND     X063  ; S6plant節流出
      OUT     T120 K5  ; 1322
3685  LD      M1322  ; 節流出
      AND     T120  ; 1322
      LD      M1323  ; 節流歸
      ANI     M1321  ; idle
      ORB
      AND     M0  ; Auto Status
      AND     X002  ; 急停
      ANI     M3110  ; S6plant節流歸異常
      ANI     M3111  ; S6plant節流出異常
      OUT     M1323  ; 節流歸
3697  LD      M1323  ; 節流歸
      SET     M44  ; S6plate有料flag
3699  LD      M1323  ; 節流歸
      ANI     X062  ; S6plant節流歸
      OUT     T410 K3000
3704  LD      T410
      SET     M3110  ; S6plant節流歸異常
3707  LD      M1322  ; 節流出
      ANI     X063  ; S6plant節流出
      OUT     T411 K3000
3712  LD      T411
      SET     M3111  ; S6plant節流出異常
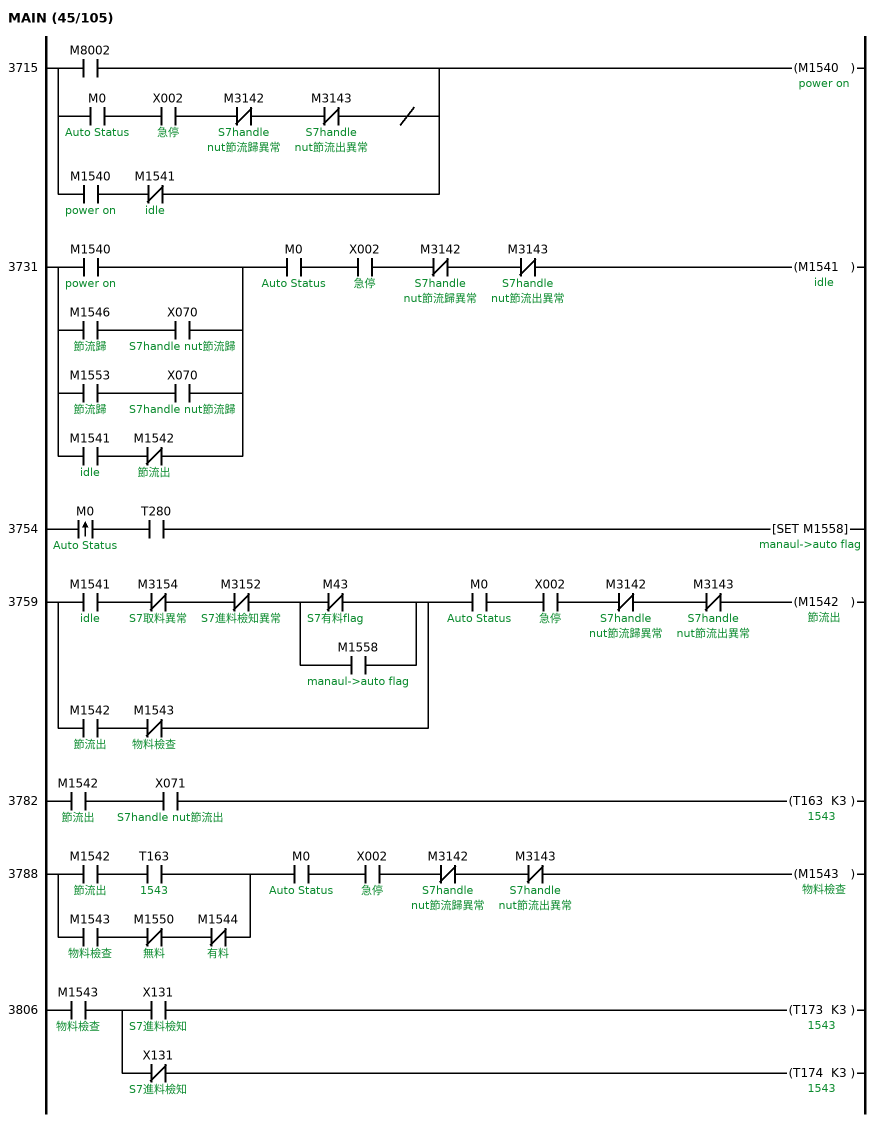
3715  LD      M8002
      LD      M0  ; Auto Status
      AND     X002  ; 急停
      ANI     M3142  ; S7handle nut節流歸異常
      ANI     M3143  ; S7handle nut節流出異常
      INV
      ORB
      LD      M1540  ; power on
      ANI     M1541  ; idle
      ORB
      OUT     M1540  ; power on
3731  LD      M1540  ; power on
      LD      M1546  ; 節流歸
      AND     X070  ; S7handle nut節流歸
      ORB
      LD      M1553  ; 節流歸
      AND     X070  ; S7handle nut節流歸
      ORB
      LD      M1541  ; idle
      ANI     M1542  ; 節流出
      ORB
      AND     M0  ; Auto Status
      AND     X002  ; 急停
      ANI     M3142  ; S7handle nut節流歸異常
      ANI     M3143  ; S7handle nut節流出異常
      OUT     M1541  ; idle
3754  LDP     M0  ; Auto Status
      AND     T280
      SET     M1558  ; manaul->auto flag
3759  LD      M1541  ; idle
      ANI     M3154  ; S7取料異常
      ANI     M3152  ; S7進料檢知異常
      LDI     M43  ; S7有料flag
      OR      M1558  ; manaul->auto flag
      ANB
      LD      M1542  ; 節流出
      ANI     M1543  ; 物料檢查
      ORB
      AND     M0  ; Auto Status
      AND     X002  ; 急停
      ANI     M3142  ; S7handle nut節流歸異常
      ANI     M3143  ; S7handle nut節流出異常
      OUT     M1542  ; 節流出
3782  LD      M1542  ; 節流出
      AND     X071  ; S7handle nut節流出
      OUT     T163 K3  ; 1543
3788  LD      M1542  ; 節流出
      AND     T163  ; 1543
      LD      M1543  ; 物料檢查
      ANI     M1550  ; 無料
      ANI     M1544  ; 有料
      ORB
      AND     M0  ; Auto Status
      AND     X002  ; 急停
      ANI     M3142  ; S7handle nut節流歸異常
      ANI     M3143  ; S7handle nut節流出異常
      OUT     M1543  ; 物料檢查
3806  LD      M1543  ; 物料檢查
      MPS
      AND     X131  ; S7進料檢知
      OUT     T173 K3  ; 1543
      MPP
      ANI     X131  ; S7進料檢知
      OUT     T174 K3  ; 1543
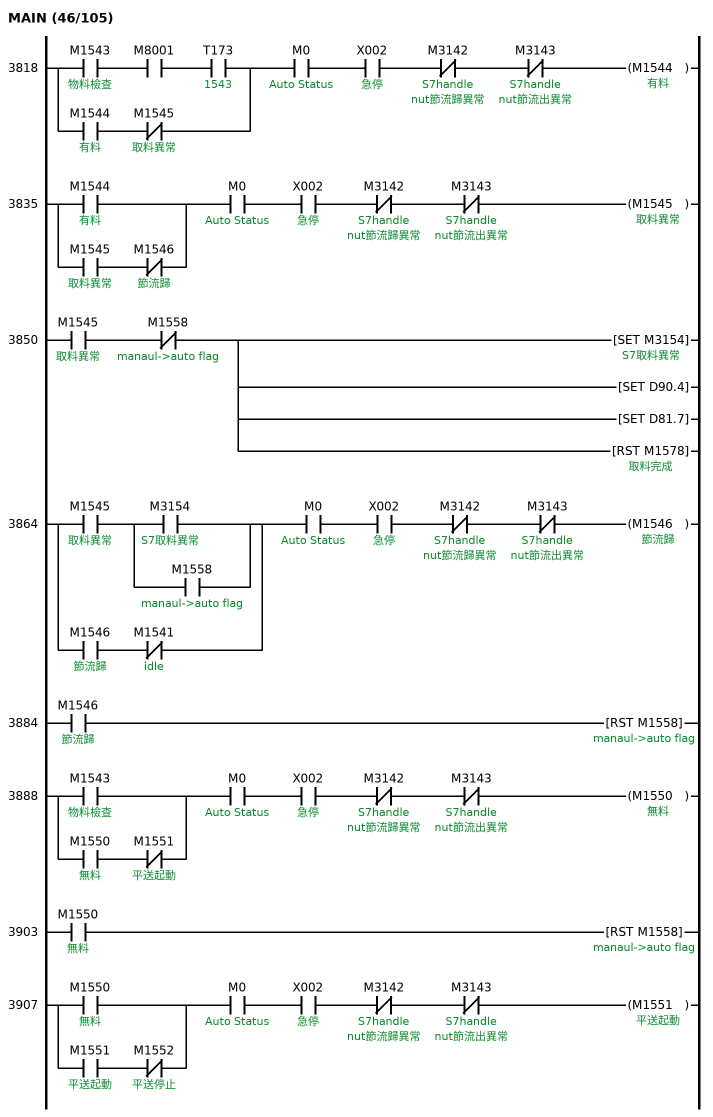
3818  LD      M1543  ; 物料檢查
      AND     M8001
      AND     T173  ; 1543
      LD      M1544  ; 有料
      ANI     M1545  ; 取料異常
      ORB
      AND     M0  ; Auto Status
      AND     X002  ; 急停
      ANI     M3142  ; S7handle nut節流歸異常
      ANI     M3143  ; S7handle nut節流出異常
      OUT     M1544  ; 有料
3835  LD      M1544  ; 有料
      LD      M1545  ; 取料異常
      ANI     M1546  ; 節流歸
      ORB
      AND     M0  ; Auto Status
      AND     X002  ; 急停
      ANI     M3142  ; S7handle nut節流歸異常
      ANI     M3143  ; S7handle nut節流出異常
      OUT     M1545  ; 取料異常
3850  LD      M1545  ; 取料異常
      ANI     M1558  ; manaul->auto flag
      SET     M3154  ; S7取料異常
      SET     D90.4
      SET     D81.7
      RST     M1578  ; 取料完成
3864  LD      M1545  ; 取料異常
      LD      M3154  ; S7取料異常
      OR      M1558  ; manaul->auto flag
      ANB
      LD      M1546  ; 節流歸
      ANI     M1541  ; idle
      ORB
      AND     M0  ; Auto Status
      AND     X002  ; 急停
      ANI     M3142  ; S7handle nut節流歸異常
      ANI     M3143  ; S7handle nut節流出異常
      OUT     M1546  ; 節流歸
3884  LD      M1546  ; 節流歸
      RST     M1558  ; manaul->auto flag
3888  LD      M1543  ; 物料檢查
      LD      M1550  ; 無料
      ANI     M1551  ; 平送起動
      ORB
      AND     M0  ; Auto Status
      AND     X002  ; 急停
      ANI     M3142  ; S7handle nut節流歸異常
      ANI     M3143  ; S7handle nut節流出異常
      OUT     M1550  ; 無料
3903  LD      M1550  ; 無料
      RST     M1558  ; manaul->auto flag
3907  LD      M1550  ; 無料
      LD      M1551  ; 平送起動
      ANI     M1552  ; 平送停止
      ORB
      AND     M0  ; Auto Status
      AND     X002  ; 急停
      ANI     M3142  ; S7handle nut節流歸異常
      ANI     M3143  ; S7handle nut節流出異常
      OUT     M1551  ; 平送起動
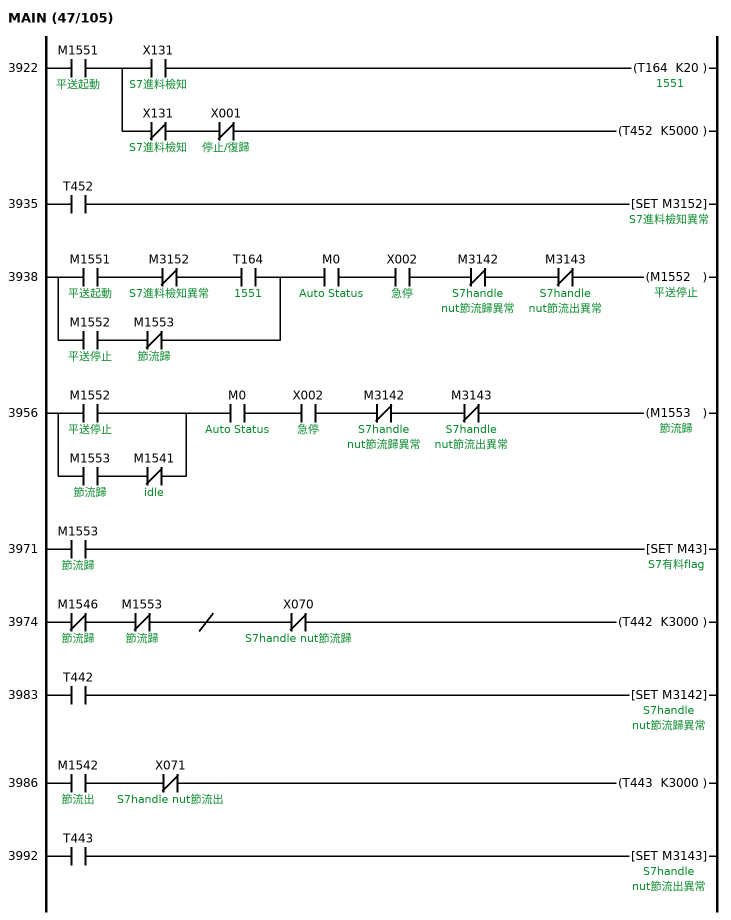
3922  LD      M1551  ; 平送起動
      MPS
      AND     X131  ; S7進料檢知
      OUT     T164 K20  ; 1551
      MPP
      ANI     X131  ; S7進料檢知
      ANI     X001  ; 停止/復歸
      OUT     T452 K5000
3935  LD      T452
      SET     M3152  ; S7進料檢知異常
3938  LD      M1551  ; 平送起動
      ANI     M3152  ; S7進料檢知異常
      AND     T164  ; 1551
      LD      M1552  ; 平送停止
      ANI     M1553  ; 節流歸
      ORB
      AND     M0  ; Auto Status
      AND     X002  ; 急停
      ANI     M3142  ; S7handle nut節流歸異常
      ANI     M3143  ; S7handle nut節流出異常
      OUT     M1552  ; 平送停止
3956  LD      M1552  ; 平送停止
      LD      M1553  ; 節流歸
      ANI     M1541  ; idle
      ORB
      AND     M0  ; Auto Status
      AND     X002  ; 急停
      ANI     M3142  ; S7handle nut節流歸異常
      ANI     M3143  ; S7handle nut節流出異常
      OUT     M1553  ; 節流歸
3971  LD      M1553  ; 節流歸
      SET     M43  ; S7有料flag
3974  LDI     M1546  ; 節流歸
      ANI     M1553  ; 節流歸
      INV
      ANI     X070  ; S7handle nut節流歸
      OUT     T442 K3000
3983  LD      T442
      SET     M3142  ; S7handle nut節流歸異常
3986  LD      M1542  ; 節流出
      ANI     X071  ; S7handle nut節流出
      OUT     T443 K3000
3992  LD      T443
      SET     M3143  ; S7handle nut節流出異常
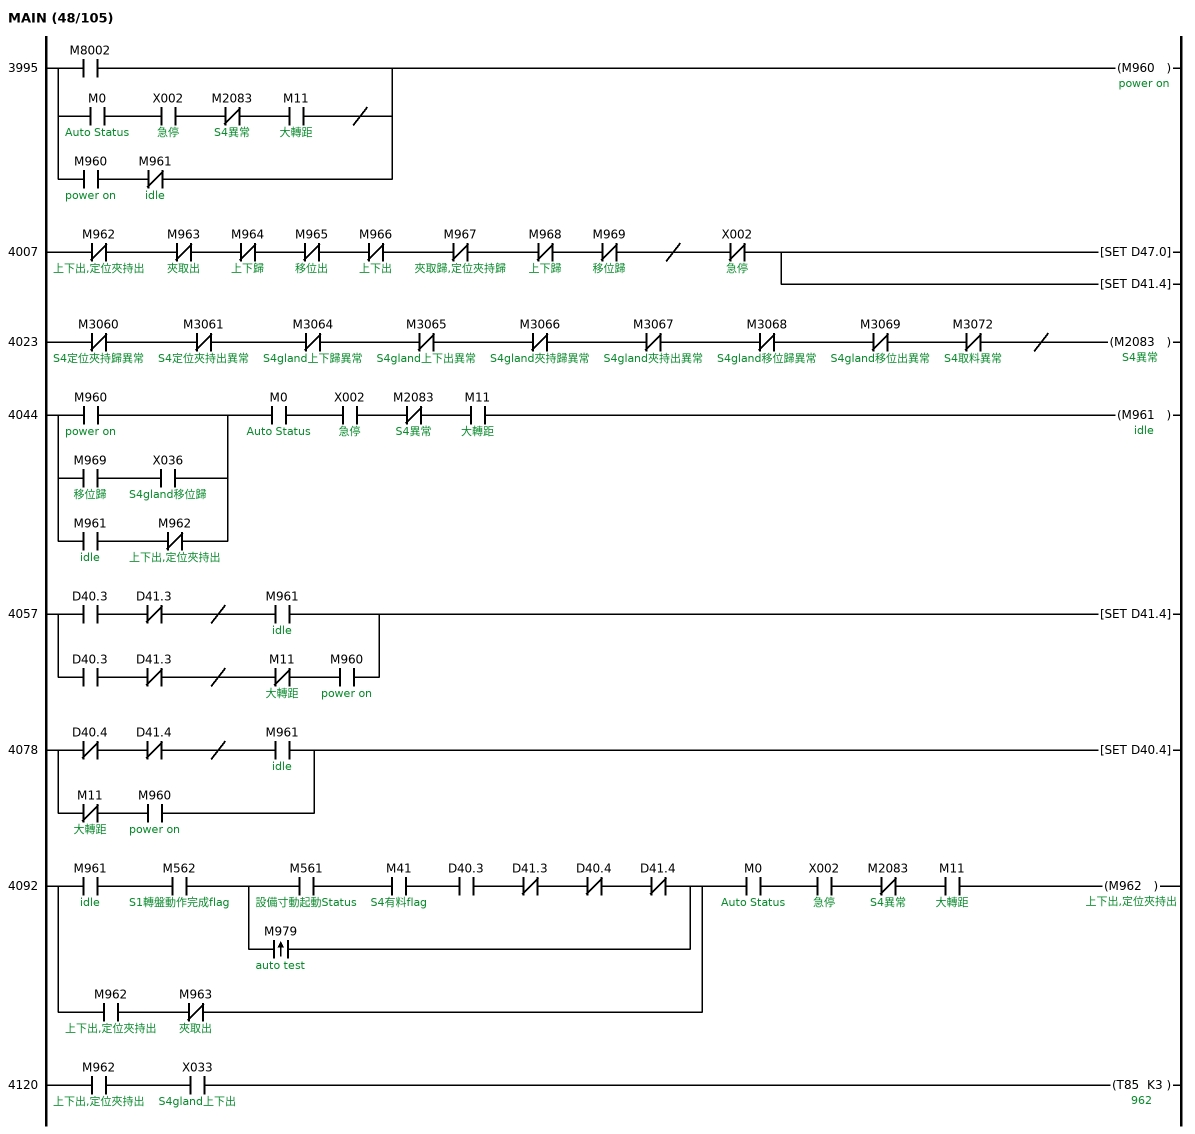
3995  LD      M8002
      LD      M0  ; Auto Status
      AND     X002  ; 急停
      ANI     M2083  ; S4異常
      AND     M11  ; 大轉距
      INV
      ORB
      LD      M960  ; power on
      ANI     M961  ; idle
      ORB
      OUT     M960  ; power on
4007  LDI     M962  ; 上下出,定位夾持出
      ANI     M963  ; 夾取出
      ANI     M964  ; 上下歸
      ANI     M965  ; 移位出
      ANI     M966  ; 上下出
      ANI     M967  ; 夾取歸,定位夾持歸
      ANI     M968  ; 上下歸
      ANI     M969  ; 移位歸
      INV
      ANI     X002  ; 急停
      SET     D47.0
      SET     D41.4
4023  LDI     M3060  ; S4定位夾持歸異常
      ANI     M3061  ; S4定位夾持出異常
      ANI     M3064  ; S4gland上下歸異常
      ANI     M3065  ; S4gland上下出異常
      ANI     M3066  ; S4gland夾持歸異常
      ANI     M3067  ; S4gland夾持出異常
      ANI     M3068  ; S4gland移位歸異常
      ANI     M3069  ; S4gland移位出異常
      ANI     M3072  ; S4取料異常
      INV
      OUT     M2083  ; S4異常
4044  LD      M960  ; power on
      LD      M969  ; 移位歸
      AND     X036  ; S4gland移位歸
      ORB
      LD      M961  ; idle
      ANI     M962  ; 上下出,定位夾持出
      ORB
      AND     M0  ; Auto Status
      AND     X002  ; 急停
      ANI     M2083  ; S4異常
      AND     M11  ; 大轉距
      OUT     M961  ; idle
4057  LD      D40.3
      ANI     D41.3
      INV
      AND     M961  ; idle
      LD      D40.3
      ANI     D41.3
      INV
      ANI     M11  ; 大轉距
      AND     M960  ; power on
      ORB
      SET     D41.4
4078  LDI     D40.4
      ANI     D41.4
      INV
      AND     M961  ; idle
      LDI     M11  ; 大轉距
      AND     M960  ; power on
      ORB
      SET     D40.4
4092  LD      M961  ; idle
      AND     M562  ; S1轉盤動作完成flag
      LD      M561  ; 設備寸動起動Status
      AND     M41  ; S4有料flag
      AND     D40.3
      ANI     D41.3
      ANI     D40.4
      ANI     D41.4
      ORP     M979  ; auto test
      ANB
      LD      M962  ; 上下出,定位夾持出
      ANI     M963  ; 夾取出
      ORB
      AND     M0  ; Auto Status
      AND     X002  ; 急停
      ANI     M2083  ; S4異常
      AND     M11  ; 大轉距
      OUT     M962  ; 上下出,定位夾持出
4120  LD      M962  ; 上下出,定位夾持出
      AND     X033  ; S4gland上下出
      OUT     T85 K3  ; 962
